# B&R Automation Studio project NAEUL004C00R13L518F00 (part 20)

#### Act_OptP0933PusherConvFB.st
```iecst
ACTION Act_OptP0933PusherConvFB:
//	IF p_bAlarmErr THEN
//		tyP0933PushConv.tyFB.tyBtnStop.bRtCompl := TRUE;
//	END_IF
	//Parameter
	diMnlMtrPshrExtSpd	:= tyP0933PushConv.tyFB.tyNumExtSpd.diValue;
//	diMnlMtrPshrExtTorq	:= tyP0933PushConv.tyFB.tyNumExtTorqPercent.diValue;

	//Pusher Torque & Force Real Time Changing
	//diMnlMtrPshrExtTorq := diConstant1 + (((tyP0933PushConv.tyFB.tyNumExtTorqPercent.diValue -10)/10)*diConstant2/100); //10~30N
//	diMnlMtrPshrExtTorq := p_tyNtParamPPTorqParam.usiStartTorque + (((tyP0933PushConv.tyFB.tyNumExtTorqPercent.diValue -10)/10)*p_tyNtParamPPTorqParam.uiRatio/100); //10~30N
	IF p_tyNtParamCurr.bProjServoPullerPusherPrep THEN
		diMnlMtrPshrExtTorq := p_tyNtParamPPTorqParam.usiStartTorque + (((tyP0933PushConv.tyFB.tyNumExtTorqPercent.diValue -10)/10)*p_tyNtParamPPTorqParam.uiRatio/100); //10~30N
	ELSE
		diMnlMtrPshrExtTorq := tyP0933PushConv.tyFB.tyNumExtTorqPercent.diValue;
	END_IF
	//Conveyor
	IF tyP0933PushConv.tyFB.tyBtnStop.bRtCompl = TRUE THEN
		diMnlPPJogSpd	:= 0;
		ePshrConvAct	:= ConvActPshrRstAll;
//		usiExtRetTest := 0; //Ah Liang

		IF p_ePshrConvStat = ConvActPshrRstAll AND p_ePshrConvStatus = Done THEN
			ePshrConvAct	:= ConvActIdle;

			tyP0933PushConv.tyFB.tyBtnEnt.bRtCompl		:= FALSE;
			tyP0933PushConv.tyFB.tyBtnEnt.bValue		:= FALSE;
			tyP0933PushConv.tyFB.tyBtnEnt.bRtLk			:= FALSE;

			tyP0933PushConv.tyFB.tyBtnExit.bRtCompl		:= FALSE;
			tyP0933PushConv.tyFB.tyBtnExit.bValue		:= FALSE;
			tyP0933PushConv.tyFB.tyBtnExit.bRtLk		:= FALSE;

			tyP0933PushConv.tyFB.tyBtnCylExit.bRtCompl	:= FALSE;
			tyP0933PushConv.tyFB.tyBtnCylExit.bValue	:= FALSE;
			tyP0933PushConv.tyFB.tyBtnCylExit.bRtLk		:= FALSE;

			tyP0933PushConv.tyFB.tyBtnStop.bRtCompl		:= FALSE;
			tyP0933PushConv.tyFB.tyBtnStop.bValue		:= TRUE;
			tyP0933PushConv.tyFB.tyBtnStop.bRtLk		:= TRUE;
		END_IF

	ELSIF tyP0933PushConv.tyFB.tyBtnEnt.bRtCompl = TRUE THEN
		tyP0933PushConv.tyFB.tyBtnEnt.bValue	:= TRUE;
		tyP0933PushConv.tyFB.tyBtnEnt.bRtLk		:= TRUE;

		tyP0933PushConv.tyFB.tyBtnStop.bValue	:= FALSE;
		tyP0933PushConv.tyFB.tyBtnStop.bRtLk	:= FALSE;

		ePshrConvAct	:= ConvActEnt;
		fUIInRtStatOff(ADR(tyP0930MagConv1.tyCom.tyBtnSwitch.uiMaskRtStat));

		IF p_ePshrConvStat = ConvActEnt AND p_ePshrConvStatus = Done THEN
			ePshrConvAct	:= ConvActIdle;

			tyP0933PushConv.tyFB.tyBtnEnt.bRtCompl	:= FALSE;

			tyP0933PushConv.tyFB.tyBtnEnt.bValue	:= FALSE;
			tyP0933PushConv.tyFB.tyBtnEnt.bRtLk		:= FALSE;

			tyP0933PushConv.tyFB.tyBtnStop.bValue	:= TRUE;
			tyP0933PushConv.tyFB.tyBtnStop.bRtLk	:= TRUE;
			fUIInRtStatHide(ADR(tyP0930MagConv1.tyCom.tyBtnSwitch.uiMaskRtStat));
		END_IF

	ELSIF tyP0933PushConv.tyFB.tyBtnExit.bRtCompl = TRUE THEN
		tyP0933PushConv.tyFB.tyBtnExit.bValue	:= TRUE;
		tyP0933PushConv.tyFB.tyBtnExit.bRtLk	:= TRUE;

		tyP0933PushConv.tyFB.tyBtnStop.bValue	:= FALSE;
		tyP0933PushConv.tyFB.tyBtnStop.bRtLk	:= FALSE;

		ePshrConvAct	:= ConvActExit;

		IF p_ePshrConvStat = ConvActExit AND p_ePshrConvStatus = Done THEN
			ePshrConvAct	:= ConvActIdle;

			tyP0933PushConv.tyFB.tyBtnExit.bRtCompl	:= FALSE;

			tyP0933PushConv.tyFB.tyBtnExit.bValue	:= FALSE;
			tyP0933PushConv.tyFB.tyBtnExit.bRtLk	:= FALSE;

			tyP0933PushConv.tyFB.tyBtnStop.bValue	:= TRUE;
			tyP0933PushConv.tyFB.tyBtnStop.bRtLk	:= TRUE;
		END_IF

	ELSIF tyP0933PushConv.tyFB.tyBtnCylExit.bRtCompl = TRUE THEN
		tyP0933PushConv.tyFB.tyBtnCylExit.bValue	:= TRUE;
		tyP0933PushConv.tyFB.tyBtnCylExit.bRtLk		:= TRUE;

		tyP0933PushConv.tyFB.tyBtnStop.bValue		:= FALSE;
		tyP0933PushConv.tyFB.tyBtnStop.bRtLk		:= FALSE;
		diMnlPPJogSpd	:= diMnlMtrPshrExtSpd*diMnlServoMtrMaxPulRatio;
		ePshrConvAct	:= ConvActExitPshr;
		fUIInRtStatOff(ADR(tyP0933PushConv.tyCom.tyBtnSwitch.uiMaskRtStat));

		IF p_ePshrConvStat = ConvActExitPshr AND p_ePshrConvStatus = Done THEN
			ePshrConvAct	:= ConvActIdle;

			tyP0933PushConv.tyFB.tyBtnCylExit.bRtCompl	:= FALSE;

			tyP0933PushConv.tyFB.tyBtnCylExit.bValue	:= FALSE;
			tyP0933PushConv.tyFB.tyBtnCylExit.bRtLk		:= FALSE;

			tyP0933PushConv.tyFB.tyBtnStop.bValue		:= TRUE;
			tyP0933PushConv.tyFB.tyBtnStop.bRtLk		:= TRUE;

		END_IF

	END_IF

	//Pusher
	IF p_tyNtParamCurr.bProjServoPullerPusherPrep = TRUE AND tyP0933PushConv.tyFB.tyBtnStop.bRtCompl = FALSE THEN

		IF tyP0933PushConv.tyCom.tyBtnSwitch.bValue = FALSE THEN
			IF tyP0933PushConv.tyFB.tyBtnRet.bRtCompl = TRUE THEN
				tyP0933PushConv.tyFB.tyBtnRet.bRtCompl	:= FALSE;

				tyP0933PushConv.tyFB.tyBtnRet.bValue	:= TRUE;
				tyP0933PushConv.tyFB.tyBtnExt.bValue	:= FALSE;

			ELSIF tyP0933PushConv.tyFB.tyBtnExt.bRtCompl = TRUE THEN
				tyP0933PushConv.tyFB.tyBtnExt.bRtCompl	:= FALSE;

				tyP0933PushConv.tyFB.tyBtnExt.bValue	:= TRUE;
				tyP0933PushConv.tyFB.tyBtnRet.bValue	:= FALSE;

			END_IF

			IF tyP0933PushConv.tyFB.tyBtnRet.bValue = TRUE THEN
				ePshrConvAct	:= ConvActPshrRet;
				diMnlPPJogSpd	:= diMnlMtrPshrExtSpd*diMnlServoMtrMaxPulRatio;

				tyP0933PushConv.tyFB.tyBtnStop.bValue		:= FALSE;
				tyP0933PushConv.tyFB.tyBtnStop.bRtLk		:= FALSE;

				IF p_ePshrConvStat = ConvActPshrRet AND p_ePshrConvStatus = Done THEN
					ePshrConvAct	:= ConvActIdle;
					diMnlPPJogSpd	:= 0;
					tyP0933PushConv.tyFB.tyBtnRet.bValue	:= FALSE;

				ELSIF p_ePshrConvStatus = Error THEN
					tyP0933PushConv.tyFB.tyBtnRet.bValue	:= FALSE;
					diMnlPPJogSpd	:= 0;
				END_IF

			ELSIF tyP0933PushConv.tyFB.tyBtnExt.bValue = TRUE THEN
				ePshrConvAct	:= ConvActPshrExt;
				diMnlPPJogSpd	:= diMnlMtrPshrExtSpd*diMnlServoMtrMaxPulRatio;
				tyP0933PushConv.tyFB.tyBtnStop.bValue		:= FALSE;
				tyP0933PushConv.tyFB.tyBtnStop.bRtLk		:= FALSE;

				IF p_ePshrConvStat = ConvActPshrExt AND p_ePshrConvStatus = Done THEN
					ePshrConvAct	:= ConvActIdle;
					diMnlPPJogSpd	:= 0;
					tyP0933PushConv.tyFB.tyBtnExt.bValue := FALSE;

				ELSIF p_ePshrConvStatus = Error THEN
					tyP0933PushConv.tyFB.tyBtnExt.bValue := FALSE;
					diMnlPPJogSpd	:= 0;
				END_IF

			END_IF

			//Update Status
			tyP0933PushConv.tyDC.tyBtnRet.bValue	:= NOT p_bPshrConvPshrExtCtrl;
			tyP0933PushConv.tyDC.tyBtnExt.bValue	:= p_bPshrConvPshrExtCtrl;

		END_IF

	ELSIF p_tyNtParamCurr.bProjServoPullerPusherPrep = FALSE AND tyP0933PushConv.tyFB.tyBtnStop.bRtCompl = FALSE
		THEN
//		IF usiExtRetTest = 0 THEN //Ah Liang Start
//			fbPushRetRestTmr(IN:=FALSE);
//			fbPushExtRestTmr(IN:=FALSE);
//		ELSIF usiExtRetTest = 1 THEN
//			fbPushRetRestTmr(IN:=TRUE);
//			fbPushExtRestTmr(IN:=FALSE);
//		ELSIF usiExtRetTest = 2 THEN
//			fbPushExtRestTmr(IN:=TRUE);
//			fbPushRetRestTmr(IN:=FALSE);
//		END_IF
//		IF fbPushRetRestTmr.Q THEN
//			tyP0933PushConv.tyFB.tyBtnExt.bRtCompl := TRUE;
//		ELSIF fbPushExtRestTmr.Q  THEN
//			tyP0933PushConv.tyFB.tyBtnRet.bRtCompl := TRUE;
//		END_IF //Ah Liang End

		IF tyP0933PushConv.tyCom.tyBtnSwitch.bValue = FALSE THEN
			IF tyP0933PushConv.tyFB.tyBtnRet.bRtCompl = TRUE THEN
				tyP0933PushConv.tyFB.tyBtnRet.bRtCompl	:= FALSE;

				tyP0933PushConv.tyFB.tyBtnRet.bValue	:= TRUE;
				tyP0933PushConv.tyFB.tyBtnExt.bValue	:= FALSE;

			ELSIF tyP0933PushConv.tyFB.tyBtnExt.bRtCompl = TRUE THEN
				tyP0933PushConv.tyFB.tyBtnExt.bRtCompl	:= FALSE;

				tyP0933PushConv.tyFB.tyBtnExt.bValue	:= TRUE;
				tyP0933PushConv.tyFB.tyBtnRet.bValue	:= FALSE;

			END_IF

			IF tyP0933PushConv.tyFB.tyBtnRet.bValue = TRUE THEN
				ePshrConvAct	:= ConvActPshrRet;

				tyP0933PushConv.tyFB.tyBtnStop.bValue		:= FALSE;
				tyP0933PushConv.tyFB.tyBtnStop.bRtLk		:= FALSE;

				IF p_ePshrConvStat = ConvActPshrRet AND p_ePshrConvStatus = Done THEN
					ePshrConvAct	:= ConvActIdle;

					tyP0933PushConv.tyFB.tyBtnRet.bValue	:= FALSE;
					//for testing Ah Liang
//					tyP0933PushConv.tyFB.tyBtnExt.bRtCompl := TRUE;
//					usiExtRetTest := 1 ;

				ELSIF p_ePshrConvStatus = Error THEN
					tyP0933PushConv.tyFB.tyBtnRet.bValue	:= FALSE;

				END_IF

			ELSIF tyP0933PushConv.tyFB.tyBtnExt.bValue = TRUE THEN
				ePshrConvAct			:= ConvActPshrExt;

				tyP0933PushConv.tyFB.tyBtnStop.bValue		:= FALSE;
				tyP0933PushConv.tyFB.tyBtnStop.bRtLk		:= FALSE;

				IF p_ePshrConvStat = ConvActPshrExt AND p_ePshrConvStatus = Done THEN
					ePshrConvAct	:= ConvActIdle;

					tyP0933PushConv.tyFB.tyBtnExt.bValue := FALSE;
					//for testing Ah Liang
//					tyP0933PushConv.tyFB.tyBtnRet.bRtCompl := TRUE;
//					usiExtRetTest := 2;
				ELSIF p_ePshrConvStatus = Error THEN
					tyP0933PushConv.tyFB.tyBtnExt.bValue := FALSE;

				END_IF

			END_IF

			//Update Status
			tyP0933PushConv.tyDC.tyBtnRet.bValue	:= NOT p_bPshrConvPshrExtCtrl;
			tyP0933PushConv.tyDC.tyBtnExt.bValue	:= p_bPshrConvPshrExtCtrl;

		END_IF

	ELSE

		tyP0933PushConv.tyFB.tyBtnExt.bRtCompl		:= FALSE;
		tyP0933PushConv.tyFB.tyBtnExt.bValue		:= FALSE;
		tyP0933PushConv.tyFB.tyBtnExt.bRtLk			:= FALSE;

		tyP0933PushConv.tyFB.tyBtnRet.bRtCompl		:= FALSE;
		tyP0933PushConv.tyFB.tyBtnRet.bValue		:= FALSE;
		tyP0933PushConv.tyFB.tyBtnRet.bRtLk			:= FALSE;

	END_IF

	//Pusher
	IF tyP0933PushConv.tyCom.tyBtnSwitch.bValue = FALSE THEN

		IF tyP0933PushConv.tyFB.tyBtnRet.bRtCompl = TRUE THEN
			tyP0933PushConv.tyFB.tyBtnRet.bRtCompl	:= FALSE;

			tyP0933PushConv.tyFB.tyBtnRet.bValue	:= TRUE;
			tyP0933PushConv.tyFB.tyBtnExt.bValue	:= FALSE;

		ELSIF tyP0933PushConv.tyFB.tyBtnExt.bRtCompl = TRUE THEN
			tyP0933PushConv.tyFB.tyBtnExt.bRtCompl	:= FALSE;

			tyP0933PushConv.tyFB.tyBtnExt.bValue	:= TRUE;
			tyP0933PushConv.tyFB.tyBtnRet.bValue	:= FALSE;

		END_IF

		IF tyP0933PushConv.tyFB.tyBtnRet.bValue = TRUE THEN
			ePshrConvAct	:= ConvActPshrRet;

			IF p_ePshrConvStat = ConvActPshrRet AND p_ePshrConvStatus = Done THEN
				ePshrConvAct	:= ConvActIdle;

				tyP0933PushConv.tyFB.tyBtnRet.bValue	:= FALSE;

			ELSIF p_ePshrConvStatus = Error THEN
				tyP0933PushConv.tyFB.tyBtnRet.bValue	:= FALSE;

			END_IF

		ELSIF tyP0933PushConv.tyFB.tyBtnExt.bValue = TRUE THEN
			ePshrConvAct	:= ConvActPshrExt;

			IF p_ePshrConvStat = ConvActPshrExt AND p_ePshrConvStatus = Done THEN
				ePshrConvAct	:= ConvActIdle;

				tyP0933PushConv.tyFB.tyBtnExt.bValue := FALSE;

			ELSIF p_ePshrConvStatus = Error THEN
				tyP0933PushConv.tyFB.tyBtnExt.bValue := FALSE;

			END_IF

		END_IF

		//Update Status
		tyP0933PushConv.tyDC.tyBtnRet.bValue	:= NOT p_bPshrConvPshrExtCtrl;
		tyP0933PushConv.tyDC.tyBtnExt.bValue	:= p_bPshrConvPshrExtCtrl;

	END_IF

	//Mask
	IF p_ePshrConvStatus = Error THEN

		fUIInRtStatOff(ADR(tyP0933PushConv.tyFB.tyBtnEnt.uiMaskRtStat));
		fUIInRtStatOff(ADR(tyP0933PushConv.tyFB.tyBtnExit.uiMaskRtStat));
		fUIInRtStatOff(ADR(tyP0933PushConv.tyFB.tyBtnExt.uiMaskRtStat));
		fUIInRtStatOff(ADR(tyP0933PushConv.tyFB.tyBtnCylExit.uiMaskRtStat));
		fUIInRtStatOff(ADR(tyP0933PushConv.tyFB.tyBtnRet.uiMaskRtStat));
		fUIInRtStatHide(ADR(tyP0933PushConv.tyCom.tyBtnSwitch.uiMaskRtStat));

	ELSIF tyP0933PushConv.tyFB.tyBtnEnt.bRtCompl = TRUE THEN

		fUIInRtStatHide(ADR(tyP0933PushConv.tyFB.tyBtnEnt.uiMaskRtStat));
		fUIInRtStatOff(ADR(tyP0933PushConv.tyFB.tyBtnExit.uiMaskRtStat));
		fUIInRtStatOff(ADR(tyP0933PushConv.tyFB.tyBtnCylExit.uiMaskRtStat));
		fUIInRtStatOff(ADR(tyP0933PushConv.tyFB.tyBtnExt.uiMaskRtStat));
		fUIInRtStatOff(ADR(tyP0933PushConv.tyFB.tyBtnRet.uiMaskRtStat));
		fUIInRtStatOff(ADR(tyP0933PushConv.tyCom.tyBtnSwitch.uiMaskRtStat));

	ELSIF tyP0933PushConv.tyFB.tyBtnExit.bRtCompl = TRUE THEN

		fUIInRtStatOff(ADR(tyP0933PushConv.tyFB.tyBtnEnt.uiMaskRtStat));
		fUIInRtStatHide(ADR(tyP0933PushConv.tyFB.tyBtnExit.uiMaskRtStat));
		fUIInRtStatOff(ADR(tyP0933PushConv.tyFB.tyBtnCylExit.uiMaskRtStat));
		fUIInRtStatOff(ADR(tyP0933PushConv.tyFB.tyBtnExt.uiMaskRtStat));
		fUIInRtStatOff(ADR(tyP0933PushConv.tyFB.tyBtnRet.uiMaskRtStat));
		fUIInRtStatOff(ADR(tyP0933PushConv.tyCom.tyBtnSwitch.uiMaskRtStat));

	ELSIF tyP0933PushConv.tyFB.tyBtnCylExit.bRtCompl = TRUE THEN

		fUIInRtStatOff(ADR(tyP0933PushConv.tyFB.tyBtnEnt.uiMaskRtStat));
		fUIInRtStatOff(ADR(tyP0933PushConv.tyFB.tyBtnExit.uiMaskRtStat));
		fUIInRtStatHide(ADR(tyP0933PushConv.tyFB.tyBtnCylExit.uiMaskRtStat));
		fUIInRtStatOff(ADR(tyP0933PushConv.tyFB.tyBtnExt.uiMaskRtStat));
		fUIInRtStatOff(ADR(tyP0933PushConv.tyFB.tyBtnRet.uiMaskRtStat));
		fUIInRtStatOff(ADR(tyP0933PushConv.tyCom.tyBtnSwitch.uiMaskRtStat));

	ELSIF tyP0933PushConv.tyFB.tyBtnExt.bValue = TRUE OR tyP0933PushConv.tyFB.tyBtnRet.bValue = TRUE THEN

		fUIInRtStatOff(ADR(tyP0933PushConv.tyFB.tyBtnEnt.uiMaskRtStat));
		fUIInRtStatOff(ADR(tyP0933PushConv.tyFB.tyBtnExit.uiMaskRtStat));
		fUIInRtStatHide(ADR(tyP0933PushConv.tyFB.tyBtnExt.uiMaskRtStat));
		fUIInRtStatOff(ADR(tyP0933PushConv.tyFB.tyBtnCylExit.uiMaskRtStat));
		fUIInRtStatHide(ADR(tyP0933PushConv.tyFB.tyBtnRet.uiMaskRtStat));
		fUIInRtStatOff(ADR(tyP0933PushConv.tyCom.tyBtnSwitch.uiMaskRtStat));

	ELSE

		fUIInRtStatHide(ADR(tyP0933PushConv.tyFB.tyBtnEnt.uiMaskRtStat));
		fUIInRtStatHide(ADR(tyP0933PushConv.tyFB.tyBtnExit.uiMaskRtStat));
		fUIInRtStatHide(ADR(tyP0933PushConv.tyFB.tyBtnExt.uiMaskRtStat));
		fUIInRtStatHide(ADR(tyP0933PushConv.tyFB.tyBtnCylExit.uiMaskRtStat));
		fUIInRtStatHide(ADR(tyP0933PushConv.tyFB.tyBtnRet.uiMaskRtStat));
		fUIInRtStatHide(ADR(tyP0933PushConv.tyCom.tyBtnSwitch.uiMaskRtStat));

	END_IF

	IF p_tyNtParamCurr.bProjOutletShutPrep AND NOT(p_tyNtParamCurr.bProjOutletShut2Prep) AND NOT(p_tyNtParamCurr.bProjOutletShut2Prep) THEN//single shutter case
		IF p_bLifterBtmSltAPosDiff OR ((p_bTravDPosDiff AND p_bTravEPosDiff AND p_bTravFPosDiff) OR NOT(p_tyDI.bOutShutterOpenRS) )
			THEN
			fUIInRtStatOff(ADR(tyP0933PushConv.tyFB.tyBtnCylExit.uiMaskRtStat));
			fUIInRtStatOff(ADR(tyP0933PushConv.tyFB.tyBtnExit.uiMaskRtStat));
			fUIInRtStatOff(ADR(tyP0933PushConv.tyFB.tyBtnExt.uiMaskRtStat));
		END_IF
	ELSIF p_tyNtParamCurr.bProjOutletShutPrep AND p_tyNtParamCurr.bProjOutletShut2Prep AND p_tyNtParamCurr.bProjOutletShut2Prep THEN //3 shutter case
		IF p_bLifterBtmSltAPosDiff OR ((p_bTravDPosDiff OR NOT(p_tyDI.bOutShutterOpenRS) ) AND (p_bTravEPosDiff OR NOT(p_tyDI.bOutShutterOpenRS2)) AND (p_bTravFPosDiff OR NOT(p_tyDI.bOutShutterOpenRS3)))
			THEN
			fUIInRtStatOff(ADR(tyP0933PushConv.tyFB.tyBtnCylExit.uiMaskRtStat));
			fUIInRtStatOff(ADR(tyP0933PushConv.tyFB.tyBtnExit.uiMaskRtStat));
			fUIInRtStatOff(ADR(tyP0933PushConv.tyFB.tyBtnExt.uiMaskRtStat));
		END_IF
	END_IF

	//Shutter Control
	IF tyP0933PushConv.tyInOutletShutterFB.tyBtnOpen.bRtCompl = TRUE THEN
		tyP0933PushConv.tyInOutletShutterFB.tyBtnOpen.bRtCompl	:= FALSE;

		tyP0933PushConv.tyInOutletShutterFB.tyBtnOpen.bValue	:= TRUE;
		tyP0933PushConv.tyInOutletShutterFB.tyBtnClose.bValue	:= FALSE;

	ELSIF tyP0933PushConv.tyInOutletShutterFB.tyBtnClose.bRtCompl = TRUE THEN
		tyP0933PushConv.tyInOutletShutterFB.tyBtnClose.bRtCompl	:= FALSE;

		tyP0933PushConv.tyInOutletShutterFB.tyBtnClose.bValue	:= TRUE;
		tyP0933PushConv.tyInOutletShutterFB.tyBtnOpen.bValue	:= FALSE;
	END_IF

	IF tyP0933PushConv.tyInOutletShutterFB.tyBtnOpen.bValue = TRUE THEN
		eInShutterAct	:= PneuActRet;
		eOutShutterAct	:= PneuActRet;

		IF (p_eInShutterStat = PneuActRet AND p_eInShutterStatus = Done)
			AND (p_eOutShutterStat = PneuActRet AND p_eOutShutterStatus = Done)
			THEN
			eInShutterAct	:= PneuActIdle;
			eOutShutterAct	:= PneuActIdle;
			tyP0933PushConv.tyInOutletShutterFB.tyBtnOpen.bValue	:= FALSE;
		ELSIF p_eInShutterStatus = Error OR p_eOutShutterStatus = Error THEN
			tyP0933PushConv.tyInOutletShutterFB.tyBtnOpen.bValue	:= FALSE;
		END_IF

	ELSIF tyP0933PushConv.tyInOutletShutterFB.tyBtnClose.bValue = TRUE THEN
		eInShutterAct	:= PneuActExt;
		eOutShutterAct	:= PneuActExt;
		IF (p_eInShutterStat = PneuActExt AND p_eInShutterStatus = Done)
			AND (p_eOutShutterStat = PneuActExt AND p_eOutShutterStatus = Done)
			THEN
			eInShutterAct	:= PneuActIdle;
			eOutShutterAct	:= PneuActIdle;
			tyP0933PushConv.tyInOutletShutterFB.tyBtnClose.bValue := FALSE;
		ELSIF p_eInShutterStatus = Error OR p_eOutShutterStatus = Error THEN
			tyP0933PushConv.tyInOutletShutterFB.tyBtnClose.bValue := FALSE;
		END_IF
	END_IF

END_ACTION
```

#### Act_OptP0933PusherConvFBStat.st
```iecst
ACTION Act_OptP0933PusherConvFBStat:

	tyP0933PushConv.tyFB.tyStringStat.sValue   := p_sPshrConvStatTxt;

END_ACTION
```

#### Act_OptP0933PusherConvDC.st
```iecst
ACTION Act_OptP0933PusherConvDC:

	//Conveyor
	IF tyP0933PushConv.tyDC.tyBtnStop.bRtCompl = TRUE THEN
		ePshrConvAct	:= ConvActStop;
	//	eMtrPshrAct	:= MtrPshrActStop;

		IF (p_ePshrConvStat = ConvActStop AND p_ePshrConvStatus = Done)
	//		AND	(p_eMtrPshrStat = MtrPshrActStop AND p_eMtrPshrStatus = Done)
			THEN

	//		eMtrPshrAct	:= MtrPshrActIdle;
			ePshrConvAct	:= ConvActIdle;

			tyP0933PushConv.tyDC.tyBtnStop.bRtCompl		:= FALSE;
			tyP0933PushConv.tyDC.tyBtnStop.bValue		:= TRUE;
			tyP0933PushConv.tyDC.tyBtnStop.bRtLk		:= TRUE;

			tyP0933PushConv.tyDC.tyBtnStart.bRtCompl	:= FALSE;
			tyP0933PushConv.tyDC.tyBtnStart.bValue		:= FALSE;
			tyP0933PushConv.tyDC.tyBtnStart.bRtLk		:= FALSE;
		END_IF

	ELSIF tyP0933PushConv.tyDC.tyBtnStart.bRtCompl = TRUE THEN
		tyP0933PushConv.tyDC.tyBtnStart.bValue	:= TRUE;
		tyP0933PushConv.tyDC.tyBtnStart.bRtLk	:= TRUE;

		tyP0933PushConv.tyDC.tyBtnStop.bValue	:= FALSE;
		tyP0933PushConv.tyDC.tyBtnStop.bRtLk	:= FALSE;

		ePshrConvAct	:= ConvActSetMtrSigOnOrLToR;

		IF p_ePshrConvStat = ConvActSetMtrSigOnOrLToR AND p_ePshrConvStatus = Done THEN
			ePshrConvAct	:= ConvActIdle;

			tyP0933PushConv.tyDC.tyBtnStart.bRtCompl	:= FALSE;
		END_IF

	END_IF

	//Pusher
	IF tyP0933PushConv.tyCom.tyBtnSwitch.bValue = TRUE THEN

		IF p_bPshrConvPshrTwoOutputCtrl = FALSE THEN

			IF tyP0933PushConv.tyDC.tyBtnRet.bRtCompl = TRUE THEN
				tyP0933PushConv.tyDC.tyBtnRet.bValue	:= TRUE;
				tyP0933PushConv.tyDC.tyBtnExt.bValue	:= FALSE;

				ePshrConvAct	:= ConvActPshrSetRet;

				IF p_ePshrConvStat = ConvActPshrSetRet AND p_ePshrConvStatus = Done THEN
					ePshrConvAct	:= ConvActIdle;

					tyP0933PushConv.tyDC.tyBtnRet.bRtCompl	:= FALSE;
				END_IF

			ELSIF tyP0933PushConv.tyDC.tyBtnExt.bRtCompl = TRUE THEN
				tyP0933PushConv.tyDC.tyBtnExt.bValue	:= TRUE;
				tyP0933PushConv.tyDC.tyBtnRet.bValue	:= FALSE;

				ePshrConvAct	:= ConvActPshrSetExt;

				IF p_ePshrConvStat = ConvActPshrSetExt AND p_ePshrConvStatus = Done THEN
					ePshrConvAct	:= ConvActIdle;

					tyP0933PushConv.tyDC.tyBtnExt.bRtCompl	:= FALSE;
				END_IF

			END_IF

		ELSE

			IF (tyP0933PushConv.tyDC.tyBtnRet.bRtCompl = TRUE) OR (tyP0933PushConv.tyDC.tyBtnExt.bRtCompl = TRUE) THEN
				IF (tyP0933PushConv.tyDC.tyBtnRet.bValue = TRUE) AND (tyP0933PushConv.tyDC.tyBtnExt.bValue = TRUE) THEN
					ePshrConvAct	:= ConvActPshrSetAll;

					IF p_ePshrConvStat = ConvActPshrSetAll AND p_ePshrConvStatus = Done THEN
						ePshrConvAct	:= ConvActIdle;

						tyP0933PushConv.tyDC.tyBtnRet.bRtCompl	:= FALSE;
						tyP0933PushConv.tyDC.tyBtnExt.bRtCompl	:= FALSE;
					END_IF

				ELSIF (tyP0933PushConv.tyDC.tyBtnRet.bValue = TRUE) AND (tyP0933PushConv.tyDC.tyBtnExt.bValue = FALSE) THEN
					ePshrConvAct	:= ConvActPshrSetRet;

					IF p_ePshrConvStat = ConvActPshrSetRet AND p_ePshrConvStatus = Done THEN
						ePshrConvAct	:= ConvActIdle;

						tyP0933PushConv.tyDC.tyBtnRet.bRtCompl	:= FALSE;
						tyP0933PushConv.tyDC.tyBtnExt.bRtCompl	:= FALSE;
					END_IF

				ELSIF (tyP0933PushConv.tyDC.tyBtnRet.bValue = FALSE) AND (tyP0933PushConv.tyDC.tyBtnExt.bValue = TRUE) THEN
					ePshrConvAct	:= ConvActPshrSetExt;

					IF p_ePshrConvStat = ConvActPshrSetExt AND p_ePshrConvStatus = Done THEN
						ePshrConvAct	:= ConvActIdle;

						tyP0933PushConv.tyDC.tyBtnRet.bRtCompl	:= FALSE;
						tyP0933PushConv.tyDC.tyBtnExt.bRtCompl	:= FALSE;
					END_IF

				ELSE
					ePshrConvAct	:= ConvActPshrRstAll;

					IF p_ePshrConvStat = ConvActPshrRstAll AND p_ePshrConvStatus = Done THEN
						ePshrConvAct	:= ConvActIdle;

						tyP0933PushConv.tyDC.tyBtnRet.bRtCompl	:= FALSE;
						tyP0933PushConv.tyDC.tyBtnExt.bRtCompl	:= FALSE;
					END_IF

				END_IF

			END_IF

		END_IF

		tyP0933PushConv.tyFB.tyBtnExt.bRtCompl	:= FALSE;
		tyP0933PushConv.tyFB.tyBtnExt.bValue	:= FALSE;
		tyP0933PushConv.tyFB.tyBtnRet.bRtCompl	:= FALSE;
		tyP0933PushConv.tyFB.tyBtnRet.bValue	:= FALSE;

	END_IF

	//For Motorized Puller
	IF tyP0933PushConv.tyDC.tyBtnAlarmRst.bRtCompl = TRUE THEN

		IF tyP0933PushConv.tyDC.tyBtnAlarmRst.bValue = TRUE THEN
			eMtrPshrAct	:= MtrPshrActSetAlmRst;

			IF p_eMtrPshrStat = MtrPshrActSetAlmRst AND p_eMtrPshrStatus = Done THEN
				eMtrPshrAct	:= MtrPshrActIdle;

				tyP0933PushConv.tyDC.tyBtnAlarmRst.bRtCompl	:= FALSE;
			END_IF
		ELSE
			eMtrPshrAct	:= MtrPshrActRstAlmRst;

			IF p_eMtrPshrStat = MtrPshrActRstAlmRst AND p_eMtrPshrStatus = Done THEN
				eMtrPshrAct	:= MtrPshrActIdle;

				tyP0933PushConv.tyDC.tyBtnAlarmRst.bRtCompl	:= FALSE;
			END_IF
		END_IF

	ELSIF tyP0933PushConv.tyDC.tyBtnBrake.bRtCompl = TRUE THEN

		IF tyP0933PushConv.tyDC.tyBtnBrake.bValue = TRUE THEN
			eMtrPshrAct	:= MtrPshrActSetBrake;

			IF p_eMtrPshrStat = MtrPshrActSetBrake AND p_eMtrPshrStatus = Done THEN
				eMtrPshrAct	:= MtrPshrActIdle;

				tyP0933PushConv.tyDC.tyBtnBrake.bRtCompl	:= FALSE;
			END_IF
		ELSE
			eMtrPshrAct	:= MtrPshrActRstBrake;

			IF p_eMtrPshrStat = MtrPshrActRstBrake AND p_eMtrPshrStatus = Done THEN
				eMtrPshrAct	:= MtrPshrActIdle;

				tyP0933PushConv.tyDC.tyBtnBrake.bRtCompl	:= FALSE;
			END_IF
		END_IF

	ELSIF tyP0933PushConv.tyDC.tyBtnSigOn.bRtCompl = TRUE THEN

		IF tyP0933PushConv.tyDC.tyBtnSigOn.bValue = TRUE THEN
			eMtrPshrAct	:= MtrPshrActSetSigOn;

			IF p_eMtrPshrStat = MtrPshrActSetSigOn AND p_eMtrPshrStatus = Done THEN
				eMtrPshrAct	:= MtrPshrActIdle;

				tyP0933PushConv.tyDC.tyBtnSigOn.bRtCompl	:= FALSE;
			END_IF
		ELSE
			eMtrPshrAct	:= MtrPshrActRstSigOn;

			IF p_eMtrPshrStat = MtrPshrActRstSigOn AND p_eMtrPshrStatus = Done THEN
				eMtrPshrAct	:= MtrPshrActIdle;

				tyP0933PushConv.tyDC.tyBtnSigOn.bRtCompl	:= FALSE;
			END_IF
		END_IF

	ELSIF tyP0933PushConv.tyDC.tyBtnSpdBinBit0.bRtCompl = TRUE THEN

		IF tyP0933PushConv.tyDC.tyBtnSpdBinBit0.bValue = TRUE THEN
			eMtrPshrAct	:= MtrPshrActSetSpdBit0;

			IF p_eMtrPshrStat = MtrPshrActSetSpdBit0 AND p_eMtrPshrStatus = Done THEN
				eMtrPshrAct	:= MtrPshrActIdle;

				tyP0933PushConv.tyDC.tyBtnSpdBinBit0.bRtCompl	:= FALSE;
			END_IF
		ELSE
			eMtrPshrAct	:= MtrPshrActRstSpdBit0;

			IF p_eMtrPshrStat = MtrPshrActRstSpdBit0 AND p_eMtrPshrStatus = Done THEN
				eMtrPshrAct	:= MtrPshrActIdle;

				tyP0933PushConv.tyDC.tyBtnSpdBinBit0.bRtCompl	:= FALSE;
			END_IF
		END_IF

	ELSIF tyP0933PushConv.tyDC.tyBtnSpdBinBit1.bRtCompl = TRUE THEN

		IF tyP0933PushConv.tyDC.tyBtnSpdBinBit1.bValue = TRUE THEN
			eMtrPshrAct	:= MtrPshrActSetSpdBit1;

			IF p_eMtrPshrStat = MtrPshrActSetSpdBit1 AND p_eMtrPshrStatus = Done THEN
				eMtrPshrAct	:= MtrPshrActIdle;

				tyP0933PushConv.tyDC.tyBtnSpdBinBit1.bRtCompl	:= FALSE;
			END_IF
		ELSE
			eMtrPshrAct	:= MtrPshrActRstSpdBit1;

			IF p_eMtrPshrStat = MtrPshrActRstSpdBit1 AND p_eMtrPshrStatus = Done THEN
				eMtrPshrAct	:= MtrPshrActIdle;

				tyP0933PushConv.tyDC.tyBtnSpdBinBit1.bRtCompl	:= FALSE;
			END_IF
		END_IF

	ELSIF tyP0933PushConv.tyDC.tyBtnSpdBinBit2.bRtCompl = TRUE THEN

		IF tyP0933PushConv.tyDC.tyBtnSpdBinBit2.bValue = TRUE THEN
			eMtrPshrAct	:= MtrPshrActSetSpdBit2;

			IF p_eMtrPshrStat = MtrPshrActSetSpdBit2 AND p_eMtrPshrStatus = Done THEN
				eMtrPshrAct	:= MtrPshrActIdle;

				tyP0933PushConv.tyDC.tyBtnSpdBinBit2.bRtCompl	:= FALSE;
			END_IF
		ELSE
			eMtrPshrAct	:= MtrPshrActRstSpdBit2;

			IF p_eMtrPshrStat = MtrPshrActRstSpdBit2 AND p_eMtrPshrStatus = Done THEN
				eMtrPshrAct	:= MtrPshrActIdle;

				tyP0933PushConv.tyDC.tyBtnSpdBinBit2.bRtCompl	:= FALSE;
			END_IF
		END_IF

	END_IF

	//Mask
	IF p_ePshrConvStatus = Error THEN

		fUIInRtStatOff(ADR(tyP0933PushConv.tyDC.tyBtnStart.uiMaskRtStat));
		fUIInRtStatOff(ADR(tyP0933PushConv.tyDC.tyBtnExt.uiMaskRtStat));
		fUIInRtStatOff(ADR(tyP0933PushConv.tyDC.tyBtnRet.uiMaskRtStat));

	ELSIF tyP0933PushConv.tyDC.tyBtnStart.bValue = TRUE THEN

		fUIInRtStatHide(ADR(tyP0933PushConv.tyDC.tyBtnStart.uiMaskRtStat));
		fUIInRtStatOff(ADR(tyP0933PushConv.tyDC.tyBtnExt.uiMaskRtStat));
		fUIInRtStatOff(ADR(tyP0933PushConv.tyDC.tyBtnRet.uiMaskRtStat));

	ELSE

		fUIInRtStatHide(ADR(tyP0933PushConv.tyDC.tyBtnStart.uiMaskRtStat));
		fUIInRtStatHide(ADR(tyP0933PushConv.tyDC.tyBtnExt.uiMaskRtStat));
		fUIInRtStatHide(ADR(tyP0933PushConv.tyDC.tyBtnRet.uiMaskRtStat));

	END_IF

	//Mask
	//	tyP0933PushConv.tyDC.tyBtnExt.uiMaskRtStat.0		:= NOT(p_eMtrPshrStatus = Error OR tyP0933PushConv.tyDC.tyBtnRet.bValue);
	tyP0933PushConv.tyDC.tyBtnRet.uiMaskRtStat.0		:= NOT(p_eMtrPshrStatus = Error OR tyP0933PushConv.tyDC.tyBtnExt.bValue);
	tyP0933PushConv.tyDC.tyBtnSigOn.uiMaskRtStat.0		:= NOT(p_eMtrPshrStatus = Error);
	tyP0933PushConv.tyDC.tyBtnAlarmRst.uiMaskRtStat.0	:= NOT(p_eMtrPshrStatus = Error);
	tyP0933PushConv.tyDC.tyBtnBrake.uiMaskRtStat.0		:= NOT(p_eMtrPshrStatus = Error);
	tyP0933PushConv.tyDC.tyBtnSpdBinBit0.uiMaskRtStat.0	:= NOT(p_eMtrPshrStatus = Error);
	tyP0933PushConv.tyDC.tyBtnSpdBinBit1.uiMaskRtStat.0	:= NOT(p_eMtrPshrStatus = Error);
	tyP0933PushConv.tyDC.tyBtnSpdBinBit2.uiMaskRtStat.0	:= NOT(p_eMtrPshrStatus = Error);

	IF p_bLifterBtmSltAPosDiff OR (p_bTravDPosDiff AND p_bTravEPosDiff AND p_bTravFPosDiff)
		OR p_eMtrPshrStatus = Error
		THEN
		fUIInRtStatOff(ADR(tyP0933PushConv.tyDC.tyBtnExt.uiMaskRtStat));
	END_IF

END_ACTION
```

#### Act_OptP0933PusherConvRstMnl.st
```iecst
ACTION Act_OptP0933RstMnl:

	IF EDGEPOS((bManualMod = FALSE) OR (p_ePshrConvStatus = Error) OR (p_eMtrPshrStatus = Error))  THEN

		ePshrConvAct	:= ConvActIdle;
		eMtrPshrAct	:= MtrPshrActIdle;

		//FB - Motor
		tyP0933PushConv.tyFB.tyBtnEnt.bRtCompl					:= FALSE;
		tyP0933PushConv.tyFB.tyBtnExit.bRtCompl					:= FALSE;
		tyP0933PushConv.tyFB.tyBtnCylExit.bRtCompl				:= FALSE;
		tyP0933PushConv.tyFB.tyBtnStop.bRtCompl					:= FALSE;

		tyP0933PushConv.tyFB.tyBtnEnt.bValue					:= FALSE;
		tyP0933PushConv.tyFB.tyBtnExit.bValue					:= FALSE;
		tyP0933PushConv.tyFB.tyBtnCylExit.bValue				:= FALSE;
		tyP0933PushConv.tyFB.tyBtnStop.bValue					:= TRUE;

		tyP0933PushConv.tyFB.tyBtnEnt.bRtLk						:= FALSE;
		tyP0933PushConv.tyFB.tyBtnExit.bRtLk					:= FALSE;
		tyP0933PushConv.tyFB.tyBtnCylExit.bRtLk					:= FALSE;
		tyP0933PushConv.tyFB.tyBtnStop.bRtLk					:= TRUE;

		tyP0933PushConv.tyFB.tyBtnEnt.uiMaskRtStat.0			:= TRUE;
		tyP0933PushConv.tyFB.tyBtnExit.uiMaskRtStat.0			:= TRUE;
		tyP0933PushConv.tyFB.tyBtnCylExit.uiMaskRtStat.0		:= TRUE;
		tyP0933PushConv.tyCom.tyBtnSwitch.uiMaskRtStat.0		:= TRUE;

		//FB - Pneu
		tyP0933PushConv.tyFB.tyBtnExt.bRtCompl					:= FALSE;
		tyP0933PushConv.tyFB.tyBtnRet.bRtCompl					:= FALSE;

		tyP0933PushConv.tyFB.tyBtnExt.bValue					:= FALSE;
		tyP0933PushConv.tyFB.tyBtnRet.bValue					:= FALSE;

		tyP0933PushConv.tyFB.tyBtnExt.uiMaskRtStat.0			:= TRUE;
		tyP0933PushConv.tyFB.tyBtnRet.uiMaskRtStat.0			:= TRUE;

		//DC - Motor
		tyP0933PushConv.tyDC.tyBtnStart.bRtCompl				:= FALSE;
		tyP0933PushConv.tyDC.tyBtnStop.bRtCompl					:= FALSE;

		tyP0933PushConv.tyDC.tyBtnStart.bValue					:= FALSE;
		tyP0933PushConv.tyDC.tyBtnStop.bValue					:= TRUE;

		tyP0933PushConv.tyDC.tyBtnStart.bRtLk					:= FALSE;
		tyP0933PushConv.tyDC.tyBtnStop.bRtLk					:= TRUE;

		tyP0933PushConv.tyDC.tyBtnStart.uiMaskRtStat.0			:= TRUE;
		tyP0933PushConv.tyCom.tyBtnSwitch.uiMaskRtStat.0		:= TRUE;

		//DC - Pneu
		tyP0933PushConv.tyDC.tyBtnExt.bRtCompl					:= FALSE;
		tyP0933PushConv.tyDC.tyBtnRet.bRtCompl					:= FALSE;

		tyP0933PushConv.tyDC.tyBtnExt.bValue					:= FALSE;
		tyP0933PushConv.tyDC.tyBtnRet.bValue					:= FALSE;

		tyP0933PushConv.tyDC.tyBtnExt.uiMaskRtStat.0			:= TRUE;
		tyP0933PushConv.tyDC.tyBtnRet.uiMaskRtStat.0			:= TRUE;

		//DC
		tyP0933PushConv.tyDC.tyBtnExt.bRtCompl			:= FALSE;
		tyP0933PushConv.tyDC.tyBtnRet.bRtCompl			:= FALSE;
		tyP0933PushConv.tyDC.tyBtnSpdBinBit0.bRtCompl	:= FALSE;
		tyP0933PushConv.tyDC.tyBtnSpdBinBit1.bRtCompl	:= FALSE;
		tyP0933PushConv.tyDC.tyBtnSpdBinBit2.bRtCompl	:= FALSE;
		tyP0933PushConv.tyDC.tyBtnSigOn.bRtCompl		:= FALSE;
		tyP0933PushConv.tyDC.tyBtnBrake.bRtCompl		:= FALSE;
		tyP0933PushConv.tyDC.tyBtnAlarmRst.bRtCompl		:= FALSE;

		tyP0933PushConv.tyDC.tyBtnExt.bValue			:= FALSE;
		tyP0933PushConv.tyDC.tyBtnRet.bValue			:= FALSE;
		tyP0933PushConv.tyDC.tyBtnSpdBinBit0.bValue		:= FALSE;
		tyP0933PushConv.tyDC.tyBtnSpdBinBit1.bValue		:= FALSE;
		tyP0933PushConv.tyDC.tyBtnSpdBinBit2.bValue		:= FALSE;
		tyP0933PushConv.tyDC.tyBtnSigOn.bValue			:= FALSE;
		tyP0933PushConv.tyDC.tyBtnBrake.bValue			:= FALSE;
		tyP0933PushConv.tyDC.tyBtnAlarmRst.bValue		:= FALSE;

	END_IF

	IF EDGEPOS(bManualMod = FALSE) THEN
		tyP0933PushConv.tyCom.tyBtnSwitch.bValue := FALSE;

		fUIInRtStatHide(ADR(tyP0933PushConv.tyDC.tyLyr.uiRtStat));
		fUIInRtStatOff(ADR(tyP0933PushConv.tyFB.tyLyr.uiRtStat));

	END_IF

	eInShutterAct	:= PneuActIdle;
	eOutShutterAct	:= PneuActIdle;

	tyP0933PushConv.tyInOutletShutterFB.tyBtnClose.bRtCompl	:= FALSE;
	tyP0933PushConv.tyInOutletShutterFB.tyBtnClose.bValue	:= FALSE;
	tyP0933PushConv.tyInOutletShutterFB.tyBtnOpen.bRtCompl	:= FALSE;
	tyP0933PushConv.tyInOutletShutterFB.tyBtnOpen.bValue	:= FALSE;

END_ACTION
```

#### Act_EntP0934Disp.st
```iecst
ACTION Act_EntP0934Disp:

	//Access Address
	p_tyC0001MotionStd ACCESS ADR(tyP0934AW.tyMotionStd);

	p_tyC0002FullMask ACCESS ADR(tyP0934AW.tyFullMaskHide);

	p_tyC0004Navi ACCESS ADR(tyP0934AW.tyNaviBack);

	p_tyC0005Main ACCESS ADR(tyCommon.tyMain);

	p_tyC0007Notif ACCESS ADR(tyCommon.tyNotif);

	p_tyC0008MsgBox ACCESS ADR(tyP0934AW.tyMsgBoxHide);

	p_tyC0009Info ACCESS ADR(tyCommon.tyInfo);

	p_tyP0934AW ACCESS ADR(tyP0934AW.tyAW);

	p_tyP0934InOutletShutterFB ACCESS ADR(tyP0934AW.tyInOutletShutterFB);

	//Display
	tyP0934AW.tyAW.tyNumNewWidth.diValue	:= p_tyProdRcpCurrRcp0.diWidthInUM;

	tyP0934AW.tyMotionStd.tyBtnPwr.bValue	:= p_bAWOpenPwrOn;

END_ACTION
```

#### Act_OptP0934Navi.st
```iecst
ACTION Act_OptP0934Navi:

	IF tyP0934AW.tyNaviBack.tyBtnBack.bRtCompl = TRUE THEN
		tyP0934AW.tyNaviBack.tyBtnBack.bRtCompl	:= FALSE;
		tyP0934AW.tyNaviBack.tyBtnBack.bValue	:= FALSE;

		eChgPage	:= UIP0920MtrNPneuCtrl;
	END_IF

END_ACTION
```

#### Act_OptP0934FullMask.st
```iecst
ACTION Act_OptP0934FullMask:

	IF eCurrPage = UIP0934AW THEN

		IF p_tyDI.bEStopSig = FALSE THEN
			p_tyC0002FullMask ACCESS ADR(tyP0934AW.tyFullMaskEStop);

		ELSIF p_tyDI.bCoverSWSig = FALSE THEN
			p_tyC0002FullMask ACCESS ADR(tyP0934AW.tyFullMaskCWSig);

		ELSIF p_tyDI.bSafetyRlySig = FALSE THEN
			p_tyC0002FullMask ACCESS ADR(tyP0934AW.tyFullMaskSafetyRly);

		ELSIF p_tyDI.bConvLftSen THEN
			p_tyC0002FullMask ACCESS ADR(tyP0934AW.tyFullMaskLftSenInterrupt);

		ELSIF p_tyDI.bConvMidSen THEN
			p_tyC0002FullMask ACCESS ADR(tyP0934AW.tyFullMaskMidSenInterrupt);

		ELSIF p_tyDI.bConvRgtSen THEN
			p_tyC0002FullMask ACCESS ADR(tyP0934AW.tyFullMaskRgtSenInterrupt);

		ELSIF p_tyDI.bConvClrSen THEN
			p_tyC0002FullMask ACCESS ADR(tyP0934AW.tyFullMaskClrSenInterrupt);

		ELSIF (p_tyNtParamCurr.bProjInletShutPrep AND p_tyDI.bInShutterCloseRS = FALSE) AND NOT(bBypassShutForCalib) THEN
			p_tyC0002FullMask ACCESS ADR(tyP0934AW.tyFullMaskInShutOpnInterrupt);

		ELSIF ((p_tyDI.bOutShutterCloseRS = FALSE AND p_tyNtParamCurr.bProjOutletShutPrep) OR (p_tyDI.bOutShutterCloseRS2 = FALSE AND p_tyNtParamCurr.bProjOutletShut2Prep )OR (p_tyDI.bOutShutterCloseRS3 = FALSE AND p_tyNtParamCurr.bProjOutletShut3Prep)) AND NOT(bBypassShutForCalib) THEN
//			IF p_tyNtParamCurr.bCurtainSenPrep THEN
//				IF (p_tyDI.bOutShutterCloseRS = FALSE AND p_tyNtParamCurr.bProjOutletShutPrep ) OR (p_tyDI.bOutShutterCloseRS2 = FALSE AND p_tyNtParamCurr.bProjOutletShut2Prep)OR (p_tyDI.bOutShutterCloseRS3 = FALSE AND p_tyNtParamCurr.bProjOutletShut3Prep )THEN
//					p_tyC0002FullMask ACCESS ADR(tyP0934AW.tyFullMaskOutShutOpnInterrupt);
//				END_IF
//			ELSE
//				IF p_tyDI.bOutShutterCloseRS = FALSE THEN
					p_tyC0002FullMask ACCESS ADR(tyP0934AW.tyFullMaskOutShutOpnInterrupt);
//				END_IF
//			END_IF
		ELSE
			p_tyC0002FullMask ACCESS ADR(tyP0934AW.tyFullMaskHide);

		END_IF

	END_IF

END_ACTION
```

#### Act_OptP0934FBCtrl.st
```iecst
ACTION Act_OptP0934FBCtrl:

	fbJogSlowToFastDlyTm.PT	:= T#2s;
	fbJogSlowToFastDlyTm;
	fbLmtRstTm;

	//Conveyor Sensor Interruption
	IF (p_tyDI.bConvLftSen OR p_tyDI.bConvMidSen OR p_tyDI.bConvRgtSen OR p_tyDI.bConvClrSen OR p_tyDI.bPusherRetRS = FALSE)
		AND eCurrPage = UIP0934AW
		THEN
		tyP0934AW.tyMotionStd.tyBtnStop.bRtCompl	:= TRUE;
	END_IF

//	IF EDGEPOS((p_udiAWOpenAxisErrID = 21570 OR p_udiAWOpenAxisErrID = 21571)
	IF EDGEPOS((p_bAWOpenFwdLmtSen OR p_bAWOpenRevLmtSen OR p_udiAWOpenAxisErrID = 21570 OR p_udiAWOpenAxisErrID = 21571)
		AND tyP0934AW.tyMotionStd.tyBtnJogOpen.bValue = FALSE
		AND tyP0934AW.tyMotionStd.tyBtnJogClose.bValue = FALSE)
	THEN
		fbLmtRstTm.IN	:= TRUE;
	END_IF

	IF fbLmtRstTm.Q = TRUE THEN
		tyP0934AW.tyMotionStd.tyBtnRst.bRtCompl		:= TRUE;
	END_IF

	IF (tyP0934AW.tyMotionStd.tyBtnJogOpen.bValue = FALSE AND tyP0934AW.tyMotionStd.tyBtnJogClose.bValue = FALSE) AND (p_bAWOpenJogging = TRUE) THEN
		bJogStopAW	:= TRUE;
	END_IF

	IF tyP0934AW.tyMotionStd.tyBtnStop.bRtCompl = TRUE THEN
		eAWOpenAct		:= AWActStop;

		IF p_eAWOpenStat = AWActStop AND p_eAWOpenStatus = Done THEN
			eAWOpenAct	:= AWActIdle;

			tyP0934AW.tyMotionStd.tyBtnStop.bRtCompl			:= FALSE;
			tyP0934AW.tyMotionStd.tyBtnJogOpen.bRtCompl			:= FALSE;
			tyP0934AW.tyMotionStd.tyBtnJogClose.bRtCompl		:= FALSE;
			tyP0934AW.tyMotionStd.tyBtnOrigin.bRtCompl			:= FALSE;
			tyP0934AW.tyMotionStd.tyBtnMovAbs.bRtCompl			:= FALSE;
			tyP0934AW.tyMotionStd.tyBtnMovRel.bRtCompl			:= FALSE;
			tyP0934AW.tyAW.tyBtnGo.bRtCompl						:= FALSE;

			tyP0934AW.tyMotionStd.tyBtnStop.bValue				:= TRUE;
			tyP0934AW.tyMotionStd.tyBtnJogOpen.bValue			:= FALSE;
			tyP0934AW.tyMotionStd.tyBtnJogClose.bValue			:= FALSE;
			tyP0934AW.tyMotionStd.tyBtnOrigin.bValue			:= FALSE;
			tyP0934AW.tyMotionStd.tyBtnMovAbs.bValue			:= FALSE;
			tyP0934AW.tyMotionStd.tyBtnMovRel.bValue			:= FALSE;
			tyP0934AW.tyAW.tyBtnGo.bValue						:= FALSE;

			tyP0934AW.tyMotionStd.tyBtnStop.bRtLk				:= TRUE;
			tyP0934AW.tyMotionStd.tyBtnJogOpen.bRtLk			:= FALSE;
			tyP0934AW.tyMotionStd.tyBtnJogClose.bRtLk			:= FALSE;
			tyP0934AW.tyMotionStd.tyBtnOrigin.bRtLk				:= FALSE;
			tyP0934AW.tyMotionStd.tyBtnMovAbs.bRtLk				:= FALSE;
			tyP0934AW.tyMotionStd.tyBtnMovRel.bRtLk				:= FALSE;
			tyP0934AW.tyAW.tyBtnGo.bRtLk						:= FALSE;
		END_IF

	ELSIF (tyP0934AW.tyMotionStd.tyBtnJogOpen.bRtCompl = TRUE) OR (tyP0934AW.tyMotionStd.tyBtnJogClose.bRtCompl = TRUE) OR (bJogStopAW = TRUE) THEN
		bJogSlow					:= FALSE;
		bJogFast					:= FALSE;
		fbJogSlowToFastDlyTm.IN		:= FALSE;

		eAWOpenAct		:= AWActJogStop;

		IF p_eAWOpenStat = AWActJogStop AND p_eAWOpenStatus = Done THEN
			eAWOpenAct	:= AWActIdle;

			bJogStopAW	:= FALSE;

			tyP0934AW.tyMotionStd.tyBtnStop.bRtCompl		:= FALSE;
			tyP0934AW.tyMotionStd.tyBtnJogOpen.bRtCompl		:= FALSE;
			tyP0934AW.tyMotionStd.tyBtnJogClose.bRtCompl	:= FALSE;
			tyP0934AW.tyMotionStd.tyBtnOrigin.bRtCompl		:= FALSE;
			tyP0934AW.tyMotionStd.tyBtnMovAbs.bRtCompl		:= FALSE;
			tyP0934AW.tyMotionStd.tyBtnMovRel.bRtCompl		:= FALSE;
			tyP0934AW.tyAW.tyBtnGo.bRtCompl					:= FALSE;

			tyP0934AW.tyMotionStd.tyBtnStop.bValue			:= TRUE;
			tyP0934AW.tyMotionStd.tyBtnJogOpen.bValue		:= FALSE;
			tyP0934AW.tyMotionStd.tyBtnJogClose.bValue		:= FALSE;
			tyP0934AW.tyMotionStd.tyBtnOrigin.bValue		:= FALSE;
			tyP0934AW.tyMotionStd.tyBtnMovAbs.bValue		:= FALSE;
			tyP0934AW.tyMotionStd.tyBtnMovRel.bValue		:= FALSE;
			tyP0934AW.tyAW.tyBtnGo.bValue					:= FALSE;

			tyP0934AW.tyMotionStd.tyBtnStop.bRtLk			:= TRUE;
			tyP0934AW.tyMotionStd.tyBtnJogOpen.bRtLk		:= FALSE;
			tyP0934AW.tyMotionStd.tyBtnJogClose.bRtLk		:= FALSE;
			tyP0934AW.tyMotionStd.tyBtnOrigin.bRtLk			:= FALSE;
			tyP0934AW.tyMotionStd.tyBtnMovAbs.bRtLk			:= FALSE;
			tyP0934AW.tyMotionStd.tyBtnMovRel.bRtLk			:= FALSE;
			tyP0934AW.tyAW.tyBtnGo.bRtLk					:= FALSE;
		END_IF

	ELSIF tyP0934AW.tyMotionStd.tyBtnPwr.bRtCompl = TRUE THEN
		tyP0934AW.tyMotionStd.tyBtnPwr.bRtLk					:= TRUE;

		IF tyP0934AW.tyMotionStd.tyBtnPwr.bValue = TRUE THEN
			eAWOpenAct		:= AWActPwrOn;

			IF p_eAWOpenStat = AWActPwrOn AND p_eAWOpenStatus = Done THEN
				eAWOpenAct	:= AWActIdle;

				tyP0934AW.tyMotionStd.tyBtnPwr.bRtCompl			:= FALSE;
				tyP0934AW.tyMotionStd.tyBtnPwr.bRtLk			:= FALSE;
			END_IF
		ELSE
			eAWOpenAct		:= AWActPwrOff;

			IF p_eAWOpenStat = AWActPwrOff AND p_eAWOpenStatus = Done THEN
				eAWOpenAct	:= AWActIdle;

				tyP0934AW.tyMotionStd.tyBtnPwr.bRtCompl			:= FALSE;
				tyP0934AW.tyMotionStd.tyBtnPwr.bRtLk			:= FALSE;
			END_IF
		END_IF

	ELSIF tyP0934AW.tyMotionStd.tyBtnOrigin.bRtCompl = TRUE THEN
		tyP0934AW.tyMotionStd.tyBtnOrigin.bValue				:= TRUE;
		tyP0934AW.tyMotionStd.tyBtnStop.bValue					:= FALSE;

		tyP0934AW.tyMotionStd.tyBtnOrigin.bRtLk					:= TRUE;
		tyP0934AW.tyMotionStd.tyBtnStop.bRtLk					:= FALSE;

		eAWOpenAct		:= AWActHoming;

		IF p_eAWOpenStat = AWActHoming AND p_eAWOpenStatus = Done THEN
			eAWOpenAct	:= AWActIdle;

			tyP0934AW.tyMotionStd.tyBtnOrigin.bRtCompl			:= FALSE;
			tyP0934AW.tyMotionStd.tyBtnOrigin.bValue			:= FALSE;
			tyP0934AW.tyMotionStd.tyBtnStop.bValue				:= TRUE;

			tyP0934AW.tyMotionStd.tyBtnOrigin.bRtLk				:= FALSE;
			tyP0934AW.tyMotionStd.tyBtnStop.bRtLk				:= TRUE;
		END_IF

	ELSIF tyP0934AW.tyMotionStd.tyBtnRst.bRtCompl = TRUE THEN
		tyP0934AW.tyMotionStd.tyBtnRst.bValue					:= TRUE;
		tyP0934AW.tyMotionStd.tyBtnRst.bRtLk					:= TRUE;

		eAWOpenAct		:= AWActRstAxisErr;

		IF p_eAWOpenStat = AWActRstAxisErr AND p_eAWOpenStatus = Done THEN
			eAWOpenAct	:= AWActIdle;

			tyP0934AW.tyMotionStd.tyBtnRst.bRtCompl				:= FALSE;
			tyP0934AW.tyMotionStd.tyBtnRst.bValue				:= FALSE;
			tyP0934AW.tyMotionStd.tyBtnRst.bRtLk				:= FALSE;

			fbLmtRstTm.IN			:= FALSE;
		END_IF

	ELSIF tyP0934AW.tyAW.tyBtnGo.bRtCompl = TRUE THEN
		tyP0934AW.tyAW.tyBtnGo.bValue							:= TRUE;
		tyP0934AW.tyMotionStd.tyBtnStop.bValue					:= FALSE;

		tyP0934AW.tyAW.tyBtnGo.bRtLk							:= TRUE;
		tyP0934AW.tyMotionStd.tyBtnStop.bRtLk					:= FALSE;

		diMnlAWGoWidth		:= tyP0934AW.tyAW.tyNumNewWidth.diValue;
		diMnlAWNomSpd		:= tyP0934AW.tyMotionStd.tyNumNomSpd.diValue;

		eAWOpenAct		:= AWActGoWidth;

		IF p_eAWOpenStat = AWActGoWidth AND p_eAWOpenStatus = Done THEN
			eAWOpenAct	:= AWActIdle;

			tyP0934AW.tyAW.tyBtnGo.bRtCompl						:= FALSE;
			tyP0934AW.tyAW.tyBtnGo.bValue						:= FALSE;
			tyP0934AW.tyMotionStd.tyBtnStop.bValue				:= TRUE;

			tyP0934AW.tyAW.tyBtnGo.bRtLk						:= FALSE;
			tyP0934AW.tyMotionStd.tyBtnStop.bRtLk				:= TRUE;
		END_IF

	ELSIF tyP0934AW.tyMotionStd.tyBtnMovAbs.bRtCompl = TRUE THEN
		tyP0934AW.tyMotionStd.tyBtnMovAbs.bValue				:= TRUE;
		tyP0934AW.tyMotionStd.tyBtnStop.bValue					:= FALSE;

		tyP0934AW.tyMotionStd.tyBtnMovAbs.bRtLk					:= TRUE;
		tyP0934AW.tyMotionStd.tyBtnStop.bRtLk					:= FALSE;

		diMnlAWTargetPos	:= tyP0934AW.tyMotionStd.tyNumTargetPos.diValue;
		diMnlAWNomSpd		:= tyP0934AW.tyMotionStd.tyNumNomSpd.diValue;

		eAWOpenAct		:= AWActMovAbs;

		IF p_eAWOpenStat = AWActMovAbs AND p_eAWOpenStatus = Done THEN
			eAWOpenAct	:= AWActIdle;

			tyP0934AW.tyMotionStd.tyBtnMovAbs.bRtCompl			:= FALSE;
			tyP0934AW.tyMotionStd.tyBtnMovAbs.bValue			:= FALSE;
			tyP0934AW.tyMotionStd.tyBtnStop.bValue				:= TRUE;

			tyP0934AW.tyMotionStd.tyBtnMovAbs.bRtLk				:= FALSE;
			tyP0934AW.tyMotionStd.tyBtnStop.bRtLk				:= TRUE;
		END_IF

	ELSIF tyP0934AW.tyMotionStd.tyBtnMovRel.bRtCompl = TRUE THEN
		tyP0934AW.tyMotionStd.tyBtnMovRel.bValue				:= TRUE;
		tyP0934AW.tyMotionStd.tyBtnStop.bValue					:= FALSE;

		tyP0934AW.tyMotionStd.tyBtnMovRel.bRtLk					:= TRUE;
		tyP0934AW.tyMotionStd.tyBtnStop.bRtLk					:= FALSE;

		diMnlAWStepSize		:= tyP0934AW.tyMotionStd.tyNumStepSize.diValue;
		diMnlAWNomSpd		:= tyP0934AW.tyMotionStd.tyNumNomSpd.diValue;

		eAWOpenAct		:= AWActMovRel;

		IF p_eAWOpenStat = AWActMovRel AND p_eAWOpenStatus = Done THEN
			eAWOpenAct	:= AWActIdle;

			tyP0934AW.tyMotionStd.tyBtnMovRel.bRtCompl			:= FALSE;
			tyP0934AW.tyMotionStd.tyBtnMovRel.bValue			:= FALSE;
			tyP0934AW.tyMotionStd.tyBtnStop.bValue				:= TRUE;

			tyP0934AW.tyMotionStd.tyBtnMovRel.bRtLk				:= FALSE;
			tyP0934AW.tyMotionStd.tyBtnStop.bRtLk				:= TRUE;
		END_IF

	ELSIF (tyP0934AW.tyMotionStd.tyBtnJogOpen.bValue = TRUE) AND (fbJogSlowToFastDlyTm.Q = FALSE) AND (bJogSlow = FALSE) THEN
		tyP0934AW.tyMotionStd.tyBtnStop.bValue					:= FALSE;
		tyP0934AW.tyMotionStd.tyBtnStop.bRtLk					:= FALSE;

		fbJogSlowToFastDlyTm.IN		:= TRUE;

		diMnlAWJogSpd		:= tyP0934AW.tyMotionStd.tyNumSlwSpd.diValue;

		eAWOpenAct		:= AWActJogOpen;

		IF p_eAWOpenStat = AWActJogOpen AND p_eAWOpenStatus = Done THEN
			eAWOpenAct	:= AWActIdle;
			bJogSlow				:= TRUE;
		ELSIF p_eAWOpenStatus = Error THEN
			fbJogSlowToFastDlyTm.IN	:= FALSE;
			bJogSlow				:= TRUE;
		END_IF

	ELSIF (tyP0934AW.tyMotionStd.tyBtnJogOpen.bValue = TRUE) AND (fbJogSlowToFastDlyTm.Q = TRUE) AND (bJogFast = FALSE) THEN
		tyP0934AW.tyMotionStd.tyBtnStop.bValue					:= FALSE;
		tyP0934AW.tyMotionStd.tyBtnStop.bRtLk					:= FALSE;

		fbJogSlowToFastDlyTm.IN		:= TRUE;

		diMnlAWJogSpd		:= tyP0934AW.tyMotionStd.tyNumNomSpd.diValue;

		eAWOpenAct		:= AWActJogOpen;

		IF p_eAWOpenStat = AWActJogOpen AND p_eAWOpenStatus = Done THEN
			eAWOpenAct	:= AWActIdle;
			bJogFast				:= TRUE;
		ELSIF p_eAWOpenStatus = Error THEN
			fbJogSlowToFastDlyTm.IN	:= FALSE;
			bJogFast				:= TRUE;
		END_IF

	ELSIF (tyP0934AW.tyMotionStd.tyBtnJogClose.bValue = TRUE) AND (fbJogSlowToFastDlyTm.Q = FALSE) AND (bJogSlow = FALSE) THEN
		tyP0934AW.tyMotionStd.tyBtnStop.bValue					:= FALSE;
		tyP0934AW.tyMotionStd.tyBtnStop.bRtLk					:= FALSE;

		fbJogSlowToFastDlyTm.IN		:= TRUE;

		diMnlAWJogSpd		:= tyP0934AW.tyMotionStd.tyNumSlwSpd.diValue;

		eAWOpenAct		:= AWActJogClose;

		IF p_eAWOpenStat = AWActJogClose AND p_eAWOpenStatus = Done THEN
			eAWOpenAct	:= AWActIdle;
			bJogSlow				:= TRUE;
		ELSIF p_eAWOpenStatus = Error THEN
			fbJogSlowToFastDlyTm.IN	:= FALSE;
			bJogSlow				:= TRUE;
		END_IF

	ELSIF (tyP0934AW.tyMotionStd.tyBtnJogClose.bValue = TRUE) AND (fbJogSlowToFastDlyTm.Q = TRUE) AND (bJogFast = FALSE) THEN
		tyP0934AW.tyMotionStd.tyBtnStop.bValue					:= FALSE;
		tyP0934AW.tyMotionStd.tyBtnStop.bRtLk					:= FALSE;

		fbJogSlowToFastDlyTm.IN		:= TRUE;

		diMnlAWJogSpd		:= tyP0934AW.tyMotionStd.tyNumNomSpd.diValue;

		eAWOpenAct		:= AWActJogClose;

		IF p_eAWOpenStat = AWActJogClose AND p_eAWOpenStatus = Done THEN
			eAWOpenAct	:= AWActIdle;
			bJogFast				:= TRUE;
		ELSIF p_eAWOpenStatus = Error THEN
			fbJogSlowToFastDlyTm.IN	:= FALSE;
			bJogFast				:= TRUE;
		END_IF
	END_IF

	//Shutter Control
	IF tyP0934AW.tyInOutletShutterFB.tyBtnOpen.bRtCompl = TRUE THEN
		tyP0934AW.tyInOutletShutterFB.tyBtnOpen.bRtCompl	:= FALSE;

		tyP0934AW.tyInOutletShutterFB.tyBtnOpen.bValue	:= TRUE;
		tyP0934AW.tyInOutletShutterFB.tyBtnClose.bValue	:= FALSE;

	ELSIF tyP0934AW.tyInOutletShutterFB.tyBtnClose.bRtCompl = TRUE THEN
		tyP0934AW.tyInOutletShutterFB.tyBtnClose.bRtCompl	:= FALSE;

		tyP0934AW.tyInOutletShutterFB.tyBtnClose.bValue	:= TRUE;
		tyP0934AW.tyInOutletShutterFB.tyBtnOpen.bValue	:= FALSE;
	END_IF

	IF tyP0934AW.tyInOutletShutterFB.tyBtnOpen.bValue = TRUE THEN
		eInShutterAct	:= PneuActRet;
		eOutShutterAct	:= PneuActRet;

		IF (p_eInShutterStat = PneuActRet AND p_eInShutterStatus = Done)
			AND (p_eOutShutterStat = PneuActRet AND p_eOutShutterStatus = Done)
			THEN
			eInShutterAct	:= PneuActIdle;
			eOutShutterAct	:= PneuActIdle;
			tyP0934AW.tyInOutletShutterFB.tyBtnOpen.bValue	:= FALSE;
		ELSIF p_eInShutterStatus = Error OR p_eOutShutterStatus = Error THEN
			tyP0934AW.tyInOutletShutterFB.tyBtnOpen.bValue	:= FALSE;
		END_IF

	ELSIF tyP0934AW.tyInOutletShutterFB.tyBtnClose.bValue = TRUE THEN
		eInShutterAct	:= PneuActExt;
		eOutShutterAct	:= PneuActExt;
		IF (p_eInShutterStat = PneuActExt AND p_eInShutterStatus = Done)
			AND (p_eOutShutterStat = PneuActExt AND p_eOutShutterStatus = Done)
			THEN
			eInShutterAct	:= PneuActIdle;
			eOutShutterAct	:= PneuActIdle;
			tyP0934AW.tyInOutletShutterFB.tyBtnClose.bValue := FALSE;
		ELSIF p_eInShutterStatus = Error OR p_eOutShutterStatus = Error THEN
			tyP0934AW.tyInOutletShutterFB.tyBtnClose.bValue := FALSE;
		END_IF
	END_IF

END_ACTION
```

#### Act_OptP0934FBStat.st
```iecst
ACTION Act_OptP0934FBStat:

	IF p_bAWOpenAxisErr = TRUE THEN
		tyP0934AW.tyMotionStd.tyStringStat.sValue	:= p_sAWOpenAxisErrTxt;
	ELSE
		IF NOT(p_bAWOpenJogging AND p_eAWOpenStat = AWActIdle) THEN
			tyP0934AW.tyMotionStd.tyStringStat.sValue	:= p_sAWOpenStatTxt;
		END_IF
	END_IF

END_ACTION
```

#### Act_OptP0934Mask.st
```iecst
ACTION Act_OptP0934Mask:

	// Interlock Power
	IF p_bAWOpenAxisErr = TRUE AND p_bAWOpenPwrOn = FALSE THEN
		fUIInRtStatOff(ADR(tyP0934AW.tyMotionStd.tyBtnPwr.uiMaskRtStat));
		tyP0934AW.tyMotionStd.tyBtnPwr.bValue		:= FALSE;
	ELSE
		fUIInRtStatHide(ADR(tyP0934AW.tyMotionStd.tyBtnPwr.uiMaskRtStat));
	END_IF

	// Interlock Others Move
	IF p_bAWOpenAxisErr = TRUE OR p_bAWOpenPwrOn = FALSE THEN
		fUIInRtStatOff(ADR(tyP0934AW.tyMotionStd.tyBtnOrigin.uiMaskRtStat));
		fUIInRtStatOff(ADR(tyP0934AW.tyMotionStd.tyBtnMovRel.uiMaskRtStat));
		fUIInRtStatOff(ADR(tyP0934AW.tyMotionStd.tyBtnJogOpen.uiMaskRtStat));
		fUIInRtStatOff(ADR(tyP0934AW.tyMotionStd.tyBtnJogClose.uiMaskRtStat));
	ELSE
		fUIInRtStatHide(ADR(tyP0934AW.tyMotionStd.tyBtnOrigin.uiMaskRtStat));
		fUIInRtStatHide(ADR(tyP0934AW.tyMotionStd.tyBtnMovRel.uiMaskRtStat));
		fUIInRtStatHide(ADR(tyP0934AW.tyMotionStd.tyBtnJogOpen.uiMaskRtStat));
		fUIInRtStatHide(ADR(tyP0934AW.tyMotionStd.tyBtnJogClose.uiMaskRtStat));
	END_IF

	// Interlock Move Absolute
	IF p_bAWOpenAxisErr = TRUE OR p_bAWOpenPwrOn = FALSE OR p_bAWOpenIsHomed = FALSE THEN
		fUIInRtStatOff(ADR(tyP0934AW.tyAW.tyBtnGo.uiMaskRtStat));
		fUIInRtStatOff(ADR(tyP0934AW.tyMotionStd.tyBtnMovAbs.uiMaskRtStat));
	ELSE
		fUIInRtStatHide(ADR(tyP0934AW.tyAW.tyBtnGo.uiMaskRtStat));
		fUIInRtStatHide(ADR(tyP0934AW.tyMotionStd.tyBtnMovAbs.uiMaskRtStat));
	END_IF

	//Interlock Limit Sensor
	IF tyP0934AW.tyMotionStd.tyBtnOpenLmtSen.bValue = TRUE THEN
		fUIInRtStatOff(ADR(tyP0934AW.tyMotionStd.tyBtnJogOpen.uiMaskRtStat));
	END_IF

	IF tyP0934AW.tyMotionStd.tyBtnCloseLmtSen.bValue = TRUE THEN
		fUIInRtStatOff(ADR(tyP0934AW.tyMotionStd.tyBtnJogClose.uiMaskRtStat));
	END_IF

	// Interlock When Moving
	IF tyP0934AW.tyMotionStd.tyBtnOrigin.bRtCompl = TRUE THEN
		fUIInRtStatOff(ADR(tyP0934AW.tyMotionStd.tyBtnMovAbs.uiMaskRtStat));
		fUIInRtStatOff(ADR(tyP0934AW.tyMotionStd.tyBtnMovRel.uiMaskRtStat));
		fUIInRtStatOff(ADR(tyP0934AW.tyMotionStd.tyBtnJogOpen.uiMaskRtStat));
		fUIInRtStatOff(ADR(tyP0934AW.tyMotionStd.tyBtnJogClose.uiMaskRtStat));
		fUIInRtStatOff(ADR(tyP0934AW.tyAW.tyBtnGo.uiMaskRtStat));

	ELSIF tyP0934AW.tyMotionStd.tyBtnMovAbs.bRtCompl = TRUE THEN
		fUIInRtStatOff(ADR(tyP0934AW.tyMotionStd.tyBtnOrigin.uiMaskRtStat));
		fUIInRtStatOff(ADR(tyP0934AW.tyMotionStd.tyBtnMovRel.uiMaskRtStat));
		fUIInRtStatOff(ADR(tyP0934AW.tyMotionStd.tyBtnJogOpen.uiMaskRtStat));
		fUIInRtStatOff(ADR(tyP0934AW.tyMotionStd.tyBtnJogClose.uiMaskRtStat));
		fUIInRtStatOff(ADR(tyP0934AW.tyAW.tyBtnGo.uiMaskRtStat));

	ELSIF tyP0934AW.tyMotionStd.tyBtnMovRel.bRtCompl = TRUE THEN
		fUIInRtStatOff(ADR(tyP0934AW.tyMotionStd.tyBtnOrigin.uiMaskRtStat));
		fUIInRtStatOff(ADR(tyP0934AW.tyMotionStd.tyBtnMovAbs.uiMaskRtStat));
		fUIInRtStatOff(ADR(tyP0934AW.tyMotionStd.tyBtnJogOpen.uiMaskRtStat));
		fUIInRtStatOff(ADR(tyP0934AW.tyMotionStd.tyBtnJogClose.uiMaskRtStat));
		fUIInRtStatOff(ADR(tyP0934AW.tyAW.tyBtnGo.uiMaskRtStat));

	ELSIF tyP0934AW.tyMotionStd.tyBtnJogOpen.bRtCompl = TRUE OR tyP0934AW.tyMotionStd.tyBtnJogOpen.bValue = TRUE THEN
		fUIInRtStatOff(ADR(tyP0934AW.tyMotionStd.tyBtnOrigin.uiMaskRtStat));
		fUIInRtStatOff(ADR(tyP0934AW.tyMotionStd.tyBtnMovAbs.uiMaskRtStat));
		fUIInRtStatOff(ADR(tyP0934AW.tyMotionStd.tyBtnMovRel.uiMaskRtStat));
		fUIInRtStatOff(ADR(tyP0934AW.tyMotionStd.tyBtnJogClose.uiMaskRtStat));
		fUIInRtStatOff(ADR(tyP0934AW.tyAW.tyBtnGo.uiMaskRtStat));

	ELSIF tyP0934AW.tyMotionStd.tyBtnJogClose.bRtCompl = TRUE OR tyP0934AW.tyMotionStd.tyBtnJogClose.bValue = TRUE THEN
		fUIInRtStatOff(ADR(tyP0934AW.tyMotionStd.tyBtnOrigin.uiMaskRtStat));
		fUIInRtStatOff(ADR(tyP0934AW.tyMotionStd.tyBtnMovAbs.uiMaskRtStat));
		fUIInRtStatOff(ADR(tyP0934AW.tyMotionStd.tyBtnMovRel.uiMaskRtStat));
		fUIInRtStatOff(ADR(tyP0934AW.tyMotionStd.tyBtnJogOpen.uiMaskRtStat));
		fUIInRtStatOff(ADR(tyP0934AW.tyAW.tyBtnGo.uiMaskRtStat));

	ELSIF tyP0934AW.tyAW.tyBtnGo.bRtCompl = TRUE THEN
		fUIInRtStatOff(ADR(tyP0934AW.tyMotionStd.tyBtnOrigin.uiMaskRtStat));
		fUIInRtStatOff(ADR(tyP0934AW.tyMotionStd.tyBtnMovAbs.uiMaskRtStat));
		fUIInRtStatOff(ADR(tyP0934AW.tyMotionStd.tyBtnMovRel.uiMaskRtStat));
		fUIInRtStatOff(ADR(tyP0934AW.tyMotionStd.tyBtnJogOpen.uiMaskRtStat));
		fUIInRtStatOff(ADR(tyP0934AW.tyMotionStd.tyBtnJogClose.uiMaskRtStat));

	END_IF

	//Axis Error
	IF tyP0934AW.tyMotionStd.tyBtnPwr.bRtCompl = TRUE THEN
		fUIInRtStatOff(ADR(tyP0934AW.tyMotionStd.tyBtnRst.uiMaskRtStat));
	ELSE
		fUIInRtStatHide(ADR(tyP0934AW.tyMotionStd.tyBtnRst.uiMaskRtStat));
	END_IF

END_ACTION
```

#### Act_OptP0934UpdtDat.st
```iecst
ACTION Act_OptP0934UpdtDat:

	tyP0934AW.tyMotionStd.tyNumCurrPos.diValue			:= p_diAWOpenActualPos;
	tyP0934AW.tyMotionStd.tyNumErrCode.diValue			:= UDINT_TO_DINT(p_udiAWOpenAxisErrID);
	tyP0934AW.tyMotionStd.tyBitmapPwr.usiValueIdx		:= BOOL_TO_USINT(p_bAWOpenPwrOn);
	tyP0934AW.tyMotionStd.tyBitmapRst.usiValueIdx		:= BOOL_TO_USINT(NOT p_bAWOpenAxisErr);
	tyP0934AW.tyMotionStd.tyBitmapOrigin.usiValueIdx	:= BOOL_TO_USINT(p_bAWOpenIsHomed);
	tyP0934AW.tyMotionStd.tyBtnOpenLmtSen.bValue		:= p_bAWOpenOpenSen;
	tyP0934AW.tyMotionStd.tyBtnCloseLmtSen.bValue		:= p_bAWOpenCloseSen;

	//Machine Bitmap
	IF p_bAWOpenIsHomed = TRUE THEN
		IF p_diAWOpenActualPos <= (p_tyNtParamCurr.tyProdRcpWidth.diMax / 2) THEN
			tyP0934AW.tyMotionStd.tyBitmapMc.uiValueIdx 	:= 0;
		ELSE
			tyP0934AW.tyMotionStd.tyBitmapMc.uiValueIdx 	:= 1;
		END_IF
	ELSE
		tyP0934AW.tyMotionStd.tyBitmapMc.uiValueIdx	:= 0;
	END_IF

	IF p_tyNtParamCurr.eProjMag = ULMagDual THEN
		IF p_tyNtParamCurr.bMagAutoVerifyPrep = FALSE THEN
			IF 	tyP0934AW.tyMotionStd.tyBitmapMc.uiValueIdx < 100 THEN
				tyP0934AW.tyMotionStd.tyBitmapMc.uiValueIdx	:= tyP0934AW.tyMotionStd.tyBitmapMc.uiValueIdx + 300;
			END_IF
		ELSE
			IF 	tyP0934AW.tyMotionStd.tyBitmapMc.uiValueIdx < 100 THEN
				tyP0934AW.tyMotionStd.tyBitmapMc.uiValueIdx	:= tyP0934AW.tyMotionStd.tyBitmapMc.uiValueIdx + 300;
			END_IF
		END_IF
	ELSIF p_tyNtParamCurr.eProjMag = ULMagTriple AND p_tyNtParamCurr.bMagAutoVerifyPrep = TRUE AND p_tyNtParamCurr.bProjMotorizedPusherPrep = FALSE THEN
		IF 	tyP0934AW.tyMotionStd.tyBitmapMc.uiValueIdx < 200 THEN
			tyP0934AW.tyMotionStd.tyBitmapMc.uiValueIdx	:= tyP0934AW.tyMotionStd.tyBitmapMc.uiValueIdx + 200;
		END_IF
	ELSIF p_tyNtParamCurr.eProjMag = ULMagTriple AND p_tyNtParamCurr.bMagAutoVerifyPrep = FALSE AND p_tyNtParamCurr.bProjMotorizedPusherPrep = TRUE THEN
		IF 	tyP0934AW.tyMotionStd.tyBitmapMc.uiValueIdx < 400 THEN
			tyP0934AW.tyMotionStd.tyBitmapMc.uiValueIdx	:= tyP0934AW.tyMotionStd.tyBitmapMc.uiValueIdx + 400;
		END_IF
	END_IF

END_ACTION
```

#### Act_OptP0934Keypad.st
```iecst
ACTION Act_OptP0934Keypad:

	IF fUIOutRtStatTPIsOpen(ADR(tyP0934AW.tyAW.tyNumNewWidth.uiRtStat)) = TRUE THEN
		tyProperty.tyKeypad.tyStringTitle.sKeypadTitle		:= tyP0934AW.tyAW.tyNumNewWidth.sKeypadTitle;

	ELSIF fUIOutRtStatTPIsOpen(ADR(tyP0934AW.tyMotionStd.tyNumTargetPos.uiRtStat)) = TRUE THEN
		tyProperty.tyKeypad.tyStringTitle.sKeypadTitle		:= tyP0934AW.tyMotionStd.tyNumTargetPos.sKeypadTitle;

	ELSIF fUIOutRtStatTPIsOpen(ADR(tyP0934AW.tyMotionStd.tyNumStepSize.uiRtStat)) = TRUE THEN
		tyProperty.tyKeypad.tyStringTitle.sKeypadTitle		:= tyP0934AW.tyMotionStd.tyNumStepSize.sKeypadTitle;

	ELSIF fUIOutRtStatTPIsOpen(ADR(tyP0934AW.tyMotionStd.tyNumNomSpd.uiRtStat)) = TRUE THEN
		tyProperty.tyKeypad.tyStringTitle.sKeypadTitle		:= tyP0934AW.tyMotionStd.tyNumNomSpd.sKeypadTitle;

	ELSIF fUIOutRtStatTPIsOpen(ADR(tyP0934AW.tyMotionStd.tyNumSlwSpd.uiRtStat)) = TRUE THEN
		tyProperty.tyKeypad.tyStringTitle.sKeypadTitle		:= tyP0934AW.tyMotionStd.tyNumSlwSpd.sKeypadTitle;

	END_IF

END_ACTION
```

#### Act_OptP0934RstMnl.st
```iecst
ACTION Act_OptP0934RstMnl:

	IF EDGEPOS((bManualMod = FALSE) OR (p_eAWOpenStatus = Error)) THEN

		eAWOpenAct	:= AWActIdle;

		bJogSlow				:= FALSE;
		bJogFast				:= FALSE;
		fbJogSlowToFastDlyTm.IN	:= FALSE;

		tyP0934AW.tyAW.tyBtnGo.bRtCompl					:= FALSE;
		tyP0934AW.tyAW.tyBtnGo.bValue					:= FALSE;
		tyP0934AW.tyAW.tyBtnGo.bRtLk					:= FALSE;
		tyP0934AW.tyAW.tyBtnGo.uiMaskRtStat.0			:= FALSE;

		tyP0934AW.tyMotionStd.tyBtnPwr.bRtCompl				:= FALSE;
		tyP0934AW.tyMotionStd.tyBtnStop.bRtCompl			:= FALSE;
		tyP0934AW.tyMotionStd.tyBtnOrigin.bRtCompl			:= FALSE;
		tyP0934AW.tyMotionStd.tyBtnRst.bRtCompl				:= FALSE;
		tyP0934AW.tyMotionStd.tyBtnMovAbs.bRtCompl			:= FALSE;
		tyP0934AW.tyMotionStd.tyBtnMovRel.bRtCompl			:= FALSE;
		tyP0934AW.tyMotionStd.tyBtnJogOpen.bRtCompl			:= FALSE;
		tyP0934AW.tyMotionStd.tyBtnJogClose.bRtCompl		:= FALSE;

		tyP0934AW.tyMotionStd.tyBtnPwr.bValue				:= FALSE;
		tyP0934AW.tyMotionStd.tyBtnStop.bValue				:= TRUE;
		tyP0934AW.tyMotionStd.tyBtnOrigin.bValue			:= FALSE;
		tyP0934AW.tyMotionStd.tyBtnRst.bValue				:= FALSE;
		tyP0934AW.tyMotionStd.tyBtnMovAbs.bValue			:= FALSE;
		tyP0934AW.tyMotionStd.tyBtnMovRel.bValue			:= FALSE;
		tyP0934AW.tyMotionStd.tyBtnJogOpen.bValue			:= FALSE;
		tyP0934AW.tyMotionStd.tyBtnJogClose.bValue			:= FALSE;

		tyP0934AW.tyMotionStd.tyBtnPwr.bRtLk				:= FALSE;
		tyP0934AW.tyMotionStd.tyBtnStop.bRtLk				:= TRUE;
		tyP0934AW.tyMotionStd.tyBtnOrigin.bRtLk				:= FALSE;
		tyP0934AW.tyMotionStd.tyBtnRst.bRtLk				:= FALSE;
		tyP0934AW.tyMotionStd.tyBtnMovAbs.bRtLk				:= FALSE;
		tyP0934AW.tyMotionStd.tyBtnMovRel.bRtLk				:= FALSE;
		tyP0934AW.tyMotionStd.tyBtnJogOpen.bRtLk			:= FALSE;
		tyP0934AW.tyMotionStd.tyBtnJogClose.bRtLk			:= FALSE;

		tyP0934AW.tyMotionStd.tyBtnPwr.uiMaskRtStat			:= TRUE;
		tyP0934AW.tyMotionStd.tyBtnOrigin.uiMaskRtStat		:= FALSE;
		tyP0934AW.tyMotionStd.tyBtnRst.uiMaskRtStat			:= TRUE;
		tyP0934AW.tyMotionStd.tyBtnMovAbs.uiMaskRtStat		:= FALSE;
		tyP0934AW.tyMotionStd.tyBtnMovRel.uiMaskRtStat		:= FALSE;
		tyP0934AW.tyMotionStd.tyBtnJogOpen.uiMaskRtStat		:= FALSE;
		tyP0934AW.tyMotionStd.tyBtnJogClose.uiMaskRtStat	:= FALSE;

	END_IF

	eInShutterAct	:= PneuActIdle;
	eOutShutterAct	:= PneuActIdle;

	tyP0934AW.tyInOutletShutterFB.tyBtnClose.bRtCompl	:= FALSE;
	tyP0934AW.tyInOutletShutterFB.tyBtnClose.bValue	:= FALSE;
	tyP0934AW.tyInOutletShutterFB.tyBtnOpen.bRtCompl	:= FALSE;
	tyP0934AW.tyInOutletShutterFB.tyBtnOpen.bValue	:= FALSE;

END_ACTION
```

#### Act_EntP0935Disp.st
```iecst
ACTION Act_EntP0935Disp:

	//Access Address
	p_tyC0001MotionStd ACCESS ADR(tyP0935Lifter.tyMotionStd);

	p_tyC0002FullMask ACCESS ADR(tyP0935Lifter.tyFullMaskHide);

	p_tyC0004Navi ACCESS ADR(tyP0935Lifter.tyNaviBack);

	p_tyC0005Main ACCESS ADR(tyCommon.tyMain);

	p_tyC0007Notif ACCESS ADR(tyCommon.tyNotif);

	p_tyC0008MsgBox ACCESS ADR(tyP0935Lifter.tyMsgBoxHide);

	p_tyC0009Info ACCESS ADR(tyCommon.tyInfo);

	p_tyP0935Lifter ACCESS ADR(tyP0935Lifter.tyLifter);

	p_tyP0935InOutletShutterFB ACCESS ADR(tyP0935Lifter.tyInOutletShutterFB);

	//Display
	tyP0935Lifter.tyMotionStd.tyBtnPwr.bValue	:= p_bLifterBtmPwrOn;

	tyP0935Lifter.tyLifter.tyNumNewSlt.diValueMax	:= p_tyMagRcpCurrRcp.diTtlSlt;

END_ACTION
```

#### Act_OptP0935Navi.st
```iecst
ACTION Act_OptP0935Navi:

	IF tyP0935Lifter.tyNaviBack.tyBtnBack.bRtCompl = TRUE THEN
		tyP0935Lifter.tyNaviBack.tyBtnBack.bRtCompl	:= FALSE;
		tyP0935Lifter.tyNaviBack.tyBtnBack.bValue	:= FALSE;

		eChgPage	:= UIP0920MtrNPneuCtrl;

	END_IF

END_ACTION
```

#### Act_OptP0935FullMask.st
```iecst
ACTION Act_OptP0935FullMask:

	IF eCurrPage = UIP0935Lifter THEN

		IF p_tyDI.bEStopSig = FALSE THEN
			p_tyC0002FullMask ACCESS ADR(tyP0935Lifter.tyFullMaskEStop);

		ELSIF p_tyDI.bCoverSWSig = FALSE THEN
			p_tyC0002FullMask ACCESS ADR(tyP0935Lifter.tyFullMaskCWSig);

		ELSIF p_tyDI.bSafetyRlySig = FALSE THEN
			p_tyC0002FullMask ACCESS ADR(tyP0935Lifter.tyFullMaskSafetyRly);

		ELSIF p_tyDI.bPusherExtRS = TRUE THEN
			p_tyC0002FullMask ACCESS ADR(tyP0935Lifter.tyFullMaskPshrInterrupt);
		ELSIF p_tyDI.bPusherRetRS = FALSE AND p_tyDI.bPusherRetSlwSen = FALSE  THEN
			p_tyC0002FullMask ACCESS ADR(tyP0936Trav.tyFullMaskPshrNotRetInterrupt);
		ELSIF (p_tyNtParamCurr.bProjInletShutPrep AND p_tyDI.bInShutterCloseRS = FALSE) AND NOT(bBypassShutForCalib) THEN
			p_tyC0002FullMask ACCESS ADR(tyP0935Lifter.tyFullMaskInShutOpnInterrupt);

		ELSIF ((p_tyDI.bOutShutterCloseRS = FALSE AND p_tyNtParamCurr.bProjOutletShutPrep) OR (p_tyDI.bOutShutterCloseRS2 = FALSE AND p_tyNtParamCurr.bProjOutletShut2Prep )OR (p_tyDI.bOutShutterCloseRS3 = FALSE AND p_tyNtParamCurr.bProjOutletShut3Prep)) AND NOT(bBypassShutForCalib) THEN
			IF p_tyNtParamCurr.bCurtainSenPrep THEN
				IF (p_tyDI.bOutShutterCloseRS = FALSE AND p_tyNtParamCurr.bProjOutletShutPrep) OR (p_tyDI.bOutShutterCloseRS2 = FALSE AND p_tyNtParamCurr.bProjOutletShut2Prep)OR (p_tyDI.bOutShutterCloseRS3 = FALSE AND p_tyNtParamCurr.bProjOutletShut3Prep )THEN
					p_tyC0002FullMask ACCESS ADR(tyP0935Lifter.tyFullMaskOutShutOpnInterrupt);
				END_IF
			ELSE
				IF p_tyDI.bOutShutterCloseRS = FALSE THEN
					p_tyC0002FullMask ACCESS ADR(tyP0935Lifter.tyFullMaskOutShutOpnInterrupt);
				END_IF
			END_IF

		ELSIF p_tyDI.bConvLftSen THEN
			p_tyC0002FullMask ACCESS ADR(tyP0935Lifter.tyFullMaskLftSenInterrupt);

		ELSIF p_tyDI.bConvClrSen THEN
			p_tyC0002FullMask ACCESS ADR(tyP0935Lifter.tyFullMaskClrSenInterrupt);

//		ELSIF p_tyDI.bLifterSafetyLmtSW1 = FALSE OR p_tyDI.bLifterSafetyLmtSW2 = FALSE THEN
//			p_tyC0002FullMask ACCESS ADR(tyP0935Lifter.tyFullMaskSafetyLmtSW);
//			kyumin request to hide
		ELSIF p_tyDI.bLifterTimingBeltSen = FALSE THEN
			p_tyC0002FullMask ACCESS ADR(tyP0935Lifter.tyFullMaskTimingBelt);

//		ELSIF p_tyNtParamCurr.tyDISettings.diMag1FixedClampRS <> 0 AND p_tyDI.bMag1FixedClampRS = FALSE
//			AND p_tyDI.bMagPresentSen1 THEN
//			p_tyC0002FullMask ACCESS ADR(tyP0935Lifter.tyFullMaskMagClmpInt);
		ELSE
			p_tyC0002FullMask ACCESS ADR(tyP0935Lifter.tyFullMaskHide);

		END_IF

	END_IF

END_ACTION
```

#### Act_OptP0935FBCtrl.st
```iecst
ACTION Act_OptP0935FBCtrl:

	fbJogSlowToFastDlyTm.PT	:= T#2s;
	fbJogSlowToFastDlyTm;
	fbLmtRstTm;

	//Lifter Safety Sensor Interruption
	IF EDGENEG(p_tyDI.bLifterSafetyLmtSW1 AND p_tyDI.bLifterSafetyLmtSW2 AND p_tyDI.bLifterTimingBeltSen) THEN
		tyP0935Lifter.tyMotionStd.tyBtnStop.bRtCompl	:= TRUE;
	END_IF

//	IF EDGEPOS((p_udiLifterBtmAxisErrID = 21570 OR p_udiLifterBtmAxisErrID = 21571)
	IF EDGEPOS((p_bLifterBtmFwdLmtSen OR p_bLifterBtmRevLmtSen OR p_udiLifterBtmAxisErrID = 21570 OR p_udiLifterBtmAxisErrID = 21571)
		AND tyP0935Lifter.tyMotionStd.tyBtnJogDown.bValue = FALSE
		AND tyP0935Lifter.tyMotionStd.tyBtnJogUp.bValue = FALSE)
	THEN
		fbLmtRstTm.IN				:= TRUE;
	END_IF

	IF fbLmtRstTm.Q = TRUE THEN
		tyP0935Lifter.tyMotionStd.tyBtnRst.bRtCompl		:= TRUE;
	END_IF

	IF (tyP0935Lifter.tyMotionStd.tyBtnJogUp.bValue = FALSE AND tyP0935Lifter.tyMotionStd.tyBtnJogDown.bValue = FALSE) AND (p_bLifterBtmJogging = TRUE) THEN
		bJogStopLifter	:= TRUE;
	END_IF

	IF tyP0935Lifter.tyMotionStd.tyBtnStop.bRtCompl = TRUE THEN
		eLifterBtmAct		:= LifterActStop;

		IF p_eLifterBtmStat = LifterActStop AND p_eLifterBtmStatus = Done THEN
			eLifterBtmAct	:= LifterActIdle;

			tyP0935Lifter.tyMotionStd.tyBtnStop.bRtCompl			:= FALSE;
			tyP0935Lifter.tyMotionStd.tyBtnJogDown.bRtCompl			:= FALSE;
			tyP0935Lifter.tyMotionStd.tyBtnJogUp.bRtCompl			:= FALSE;
			tyP0935Lifter.tyMotionStd.tyBtnOrigin.bRtCompl			:= FALSE;
			tyP0935Lifter.tyMotionStd.tyBtnMovAbs.bRtCompl			:= FALSE;
			tyP0935Lifter.tyMotionStd.tyBtnMovRel.bRtCompl			:= FALSE;
			tyP0935Lifter.tyLifter.tyBtnGo.bRtCompl					:= FALSE;
			tyP0935Lifter.tyLifter.tyBtnNxtSlt.bRtCompl				:= FALSE;
			tyP0935Lifter.tyLifter.tyBtnPrevSlt.bRtCompl			:= FALSE;
			tyP0935Lifter.tyLifter.tyBtnGoLaneA.bRtCompl			:= FALSE;
			tyP0935Lifter.tyLifter.tyBtnGoLaneB.bRtCompl			:= FALSE;
			tyP0935Lifter.tyLifter.tyBtnGoLaneD_G.bRtCompl			:= FALSE;
			tyP0935Lifter.tyLifter.tyBtnGoLaneE_H.bRtCompl			:= FALSE;

			tyP0935Lifter.tyMotionStd.tyBtnStop.bValue				:= TRUE;
			tyP0935Lifter.tyMotionStd.tyBtnJogDown.bValue			:= FALSE;
			tyP0935Lifter.tyMotionStd.tyBtnJogUp.bValue				:= FALSE;
			tyP0935Lifter.tyMotionStd.tyBtnOrigin.bValue			:= FALSE;
			tyP0935Lifter.tyMotionStd.tyBtnMovAbs.bValue			:= FALSE;
			tyP0935Lifter.tyMotionStd.tyBtnMovRel.bValue			:= FALSE;
			tyP0935Lifter.tyLifter.tyBtnGo.bValue					:= FALSE;
			tyP0935Lifter.tyLifter.tyBtnNxtSlt.bValue				:= FALSE;
			tyP0935Lifter.tyLifter.tyBtnPrevSlt.bValue				:= FALSE;
			tyP0935Lifter.tyLifter.tyBtnGoLaneA.bValue				:= FALSE;
			tyP0935Lifter.tyLifter.tyBtnGoLaneB.bValue				:= FALSE;
			tyP0935Lifter.tyLifter.tyBtnGoLaneD_G.bValue			:= FALSE;
			tyP0935Lifter.tyLifter.tyBtnGoLaneE_H.bValue			:= FALSE;

			tyP0935Lifter.tyMotionStd.tyBtnStop.bRtLk				:= TRUE;
			tyP0935Lifter.tyMotionStd.tyBtnJogDown.bRtLk			:= FALSE;
			tyP0935Lifter.tyMotionStd.tyBtnJogUp.bRtLk				:= FALSE;
			tyP0935Lifter.tyMotionStd.tyBtnOrigin.bRtLk				:= FALSE;
			tyP0935Lifter.tyMotionStd.tyBtnMovAbs.bRtLk				:= FALSE;
			tyP0935Lifter.tyMotionStd.tyBtnMovRel.bRtLk				:= FALSE;
			tyP0935Lifter.tyLifter.tyBtnGo.bRtLk					:= FALSE;
			tyP0935Lifter.tyLifter.tyBtnNxtSlt.bRtLk				:= FALSE;
			tyP0935Lifter.tyLifter.tyBtnPrevSlt.bRtLk				:= FALSE;
			tyP0935Lifter.tyLifter.tyBtnGoLaneA.bRtLk				:= FALSE;
			tyP0935Lifter.tyLifter.tyBtnGoLaneB.bRtLk				:= FALSE;
			tyP0935Lifter.tyLifter.tyBtnGoLaneD_G.bRtLk				:= FALSE;
			tyP0935Lifter.tyLifter.tyBtnGoLaneE_H.bRtLk				:= FALSE;

		END_IF

	ELSIF (tyP0935Lifter.tyMotionStd.tyBtnJogDown.bRtCompl = TRUE) OR (tyP0935Lifter.tyMotionStd.tyBtnJogUp.bRtCompl = TRUE) OR (bJogStopLifter = TRUE) THEN
		bJogSlow					:= FALSE;
		bJogFast					:= FALSE;
		fbJogSlowToFastDlyTm.IN		:= FALSE;

		eLifterBtmAct		:= LifterActJogStop;

		IF p_eLifterBtmStat = LifterActJogStop AND p_eLifterBtmStatus = Done THEN
			eLifterBtmAct		:= LifterActIdle;

			bJogStopLifter	:= FALSE;

			tyP0935Lifter.tyMotionStd.tyBtnStop.bRtCompl			:= FALSE;
			tyP0935Lifter.tyMotionStd.tyBtnJogDown.bRtCompl			:= FALSE;
			tyP0935Lifter.tyMotionStd.tyBtnJogUp.bRtCompl			:= FALSE;
			tyP0935Lifter.tyMotionStd.tyBtnOrigin.bRtCompl			:= FALSE;
			tyP0935Lifter.tyMotionStd.tyBtnMovAbs.bRtCompl			:= FALSE;
			tyP0935Lifter.tyMotionStd.tyBtnMovRel.bRtCompl			:= FALSE;
			tyP0935Lifter.tyLifter.tyBtnGo.bRtCompl					:= FALSE;
			tyP0935Lifter.tyLifter.tyBtnNxtSlt.bRtCompl				:= FALSE;
			tyP0935Lifter.tyLifter.tyBtnPrevSlt.bRtCompl			:= FALSE;

			tyP0935Lifter.tyMotionStd.tyBtnStop.bValue				:= TRUE;
			tyP0935Lifter.tyMotionStd.tyBtnJogDown.bValue			:= FALSE;
			tyP0935Lifter.tyMotionStd.tyBtnJogUp.bValue				:= FALSE;
			tyP0935Lifter.tyMotionStd.tyBtnOrigin.bValue			:= FALSE;
			tyP0935Lifter.tyMotionStd.tyBtnMovAbs.bValue			:= FALSE;
			tyP0935Lifter.tyMotionStd.tyBtnMovRel.bValue			:= FALSE;
			tyP0935Lifter.tyLifter.tyBtnGo.bValue					:= FALSE;
			tyP0935Lifter.tyLifter.tyBtnNxtSlt.bValue				:= FALSE;
			tyP0935Lifter.tyLifter.tyBtnPrevSlt.bValue				:= FALSE;

			tyP0935Lifter.tyMotionStd.tyBtnStop.bRtLk				:= TRUE;
			tyP0935Lifter.tyMotionStd.tyBtnJogDown.bRtLk			:= FALSE;
			tyP0935Lifter.tyMotionStd.tyBtnJogUp.bRtLk				:= FALSE;
			tyP0935Lifter.tyMotionStd.tyBtnOrigin.bRtLk				:= FALSE;
			tyP0935Lifter.tyMotionStd.tyBtnMovAbs.bRtLk				:= FALSE;
			tyP0935Lifter.tyMotionStd.tyBtnMovRel.bRtLk				:= FALSE;
			tyP0935Lifter.tyLifter.tyBtnGo.bRtLk					:= FALSE;
			tyP0935Lifter.tyLifter.tyBtnNxtSlt.bRtLk				:= FALSE;
			tyP0935Lifter.tyLifter.tyBtnPrevSlt.bRtLk				:= FALSE;

		END_IF

	ELSIF tyP0935Lifter.tyMotionStd.tyBtnPwr.bRtCompl = TRUE THEN
		tyP0935Lifter.tyMotionStd.tyBtnPwr.bRtLk					:= TRUE;

		IF tyP0935Lifter.tyMotionStd.tyBtnPwr.bValue = TRUE THEN
			eLifterBtmAct		:= LifterActPwrOn;

			IF p_eLifterBtmStat = LifterActPwrOn AND p_eLifterBtmStatus = Done THEN
				eLifterBtmAct	:= LifterActIdle;

				tyP0935Lifter.tyMotionStd.tyBtnPwr.bRtCompl		:= FALSE;
				tyP0935Lifter.tyMotionStd.tyBtnPwr.bRtLk		:= FALSE;
			END_IF
		ELSE
			eLifterBtmAct		:= LifterActPwrOff;

			IF p_eLifterBtmStat = LifterActPwrOff AND p_eLifterBtmStatus = Done THEN
				eLifterBtmAct	:= LifterActIdle;

				tyP0935Lifter.tyMotionStd.tyBtnPwr.bRtCompl		:= FALSE;
				tyP0935Lifter.tyMotionStd.tyBtnPwr.bRtLk		:= FALSE;
			END_IF
		END_IF

	ELSIF tyP0935Lifter.tyMotionStd.tyBtnOrigin.bRtCompl = TRUE THEN
		tyP0935Lifter.tyMotionStd.tyBtnOrigin.bValue				:= TRUE;
		tyP0935Lifter.tyMotionStd.tyBtnStop.bValue					:= FALSE;

		tyP0935Lifter.tyMotionStd.tyBtnOrigin.bRtLk					:= TRUE;
		tyP0935Lifter.tyMotionStd.tyBtnStop.bRtLk					:= FALSE;

		eLifterBtmAct		:= LifterActHoming;

		IF p_eLifterBtmStat = LifterActHoming AND p_eLifterBtmStatus = Done THEN
			eLifterBtmAct	:= LifterActIdle;

			tyP0935Lifter.tyMotionStd.tyBtnOrigin.bRtCompl		:= FALSE;
			tyP0935Lifter.tyMotionStd.tyBtnOrigin.bValue		:= FALSE;
			tyP0935Lifter.tyMotionStd.tyBtnStop.bValue			:= TRUE;

			tyP0935Lifter.tyMotionStd.tyBtnOrigin.bRtLk			:= FALSE;
			tyP0935Lifter.tyMotionStd.tyBtnStop.bRtLk			:= TRUE;

		END_IF

	ELSIF tyP0935Lifter.tyMotionStd.tyBtnRst.bRtCompl = TRUE THEN
		tyP0935Lifter.tyMotionStd.tyBtnRst.bValue				:= TRUE;
		tyP0935Lifter.tyMotionStd.tyBtnRst.bRtLk				:= TRUE;

		eLifterBtmAct		:= LifterActRstAxisErr;

		IF p_eLifterBtmStat = LifterActRstAxisErr AND p_eLifterBtmStatus = Done THEN
			eLifterBtmAct	:= LifterActIdle;

			tyP0935Lifter.tyMotionStd.tyBtnRst.bRtCompl			:= FALSE;
			tyP0935Lifter.tyMotionStd.tyBtnRst.bValue			:= FALSE;
			tyP0935Lifter.tyMotionStd.tyBtnRst.bRtLk			:= FALSE;

			fbLmtRstTm.IN			:= FALSE;
		END_IF

	ELSIF tyP0935Lifter.tyLifter.tyBtnGo.bRtCompl = TRUE THEN
		tyP0935Lifter.tyLifter.tyBtnGo.bValue				:= TRUE;
		tyP0935Lifter.tyMotionStd.tyBtnStop.bValue			:= FALSE;

		tyP0935Lifter.tyLifter.tyBtnGo.bRtLk				:= TRUE;
		tyP0935Lifter.tyMotionStd.tyBtnStop.bRtLk			:= FALSE;

		(*diMnlLifterMag1GoSlt	:= tyP0935Lifter.tyLifter.tyNumNewSlt.diValue;*)
		diMnlLifterNomSpd		:= tyP0935Lifter.tyMotionStd.tyNumNomSpd.diValue;

		CASE tyP0935Lifter.tyLifter.tyNumMagPos.diValue OF
			1:
				eLifterBtmAct	:= LifterActGoASltPos;
				diMnlLifterMag1GoSlt	:= tyP0935Lifter.tyLifter.tyNumNewSlt.diValue;

			2:
				eLifterBtmAct	:= LifterActGoBSltPos;
				diMnlLifterMag2GoSlt	:= tyP0935Lifter.tyLifter.tyNumNewSlt.diValue;

			3:
				eLifterBtmAct	:= LifterActGoCSltPos;
				diMnlLifterMag3GoSlt	:= tyP0935Lifter.tyLifter.tyNumNewSlt.diValue;

			4:
				eLifterBtmAct	:= LifterActGoDSltPos;
				diMnlLifterMag3GoSlt	:= tyP0935Lifter.tyLifter.tyNumNewSlt.diValue;
		END_CASE

		IF (p_eLifterBtmStat = LifterActGoASltPos
			OR p_eLifterBtmStat = LifterActGoBSltPos
			OR p_eLifterBtmStat = LifterActGoCSltPos
			OR p_eLifterBtmStat = LifterActGoDSltPos)
			AND p_eLifterBtmStatus = Done THEN
			eLifterBtmAct	:= LifterActIdle;

			tyP0935Lifter.tyLifter.tyBtnGo.bRtCompl				:= FALSE;
			tyP0935Lifter.tyLifter.tyBtnGo.bValue				:= FALSE;
			tyP0935Lifter.tyMotionStd.tyBtnStop.bValue			:= TRUE;

			tyP0935Lifter.tyLifter.tyBtnGo.bRtLk				:= FALSE;
			tyP0935Lifter.tyMotionStd.tyBtnStop.bRtLk			:= TRUE;
		END_IF

	ELSIF tyP0935Lifter.tyLifter.tyBtnNxtSlt.bRtCompl = TRUE THEN
		tyP0935Lifter.tyLifter.tyBtnNxtSlt.bValue				:= TRUE;
		tyP0935Lifter.tyMotionStd.tyBtnStop.bValue				:= FALSE;

		tyP0935Lifter.tyLifter.tyBtnNxtSlt.bRtLk				:= TRUE;
		tyP0935Lifter.tyMotionStd.tyBtnStop.bRtLk				:= FALSE;

		(*diMnlLifterMag1GoSlt	:= tyP0935Lifter.tyLifter.tyNumNewSlt.diValue;*)
		diMnlLifterNomSpd		:= tyP0935Lifter.tyMotionStd.tyNumNomSpd.diValue;

		CASE tyP0935Lifter.tyLifter.tyNumMagPos.diValue OF
			1:
				eLifterBtmAct	:= LifterActGoNxtASltPos;
				diMnlLifterMag1GoSlt	:= tyP0935Lifter.tyLifter.tyNumNewSlt.diValue;
			2:
				eLifterBtmAct	:= LifterActGoNxtBSltPos;
				diMnlLifterMag2GoSlt	:= tyP0935Lifter.tyLifter.tyNumNewSlt.diValue;
			3:
				eLifterBtmAct	:= LifterActGoNxtCSltPos;
				diMnlLifterMag3GoSlt	:= tyP0935Lifter.tyLifter.tyNumNewSlt.diValue;
			4:
				eLifterBtmAct	:= LifterActGoNxtDSltPos;
		//		diMnlLifterMag4GoSlt	:= tyP0935Lifter.tyLifter.tyNumNewSlt.diValue;

		END_CASE

		IF (p_eLifterBtmStat = LifterActGoNxtASltPos
			OR p_eLifterBtmStat = LifterActGoNxtBSltPos
			OR p_eLifterBtmStat = LifterActGoNxtCSltPos
			OR p_eLifterBtmStat = LifterActGoNxtDSltPos)
			AND p_eLifterBtmStatus = Done THEN
			eLifterBtmAct	:= LifterActIdle;

			tyP0935Lifter.tyLifter.tyBtnNxtSlt.bRtCompl				:= FALSE;
			tyP0935Lifter.tyLifter.tyBtnNxtSlt.bValue				:= FALSE;
			tyP0935Lifter.tyMotionStd.tyBtnStop.bValue				:= TRUE;

			tyP0935Lifter.tyLifter.tyBtnNxtSlt.bRtLk				:= FALSE;
			tyP0935Lifter.tyMotionStd.tyBtnStop.bRtLk				:= TRUE;
		END_IF

	ELSIF tyP0935Lifter.tyLifter.tyBtnPrevSlt.bRtCompl = TRUE THEN
		tyP0935Lifter.tyLifter.tyBtnPrevSlt.bValue				:= TRUE;
		tyP0935Lifter.tyMotionStd.tyBtnStop.bValue				:= FALSE;

		tyP0935Lifter.tyLifter.tyBtnPrevSlt.bRtLk				:= TRUE;
		tyP0935Lifter.tyMotionStd.tyBtnStop.bRtLk				:= FALSE;

	//	diMnlLifterMag1GoSlt	:= tyP0935Lifter.tyLifter.tyNumNewSlt.diValue;
		diMnlLifterNomSpd		:= tyP0935Lifter.tyMotionStd.tyNumNomSpd.diValue;

		CASE tyP0935Lifter.tyLifter.tyNumMagPos.diValue OF

			1:
				eLifterBtmAct	:= LifterActGoPrevASltPos;
				diMnlLifterMag1GoSlt	:= tyP0935Lifter.tyLifter.tyNumNewSlt.diValue;

			2:
				eLifterBtmAct	:= LifterActGoPrevBSltPos;
				diMnlLifterMag2GoSlt	:= tyP0935Lifter.tyLifter.tyNumNewSlt.diValue;

			3:
				eLifterBtmAct	:= LifterActGoPrevCSltPos;
				diMnlLifterMag3GoSlt	:= tyP0935Lifter.tyLifter.tyNumNewSlt.diValue;

			4:
				eLifterBtmAct	:= LifterActGoPrevDSltPos;
		//		diMnlLifterMag4GoSlt	:= tyP0935Lifter.tyLifter.tyNumNewSlt.diValue;

		END_CASE

		IF (p_eLifterBtmStat = LifterActGoPrevASltPos
			OR p_eLifterBtmStat = LifterActGoPrevBSltPos
			OR p_eLifterBtmStat = LifterActGoPrevCSltPos
			OR p_eLifterBtmStat = LifterActGoPrevDSltPos)
			AND p_eLifterBtmStatus = Done THEN
			eLifterBtmAct	:= LifterActIdle;

			tyP0935Lifter.tyLifter.tyBtnPrevSlt.bRtCompl				:= FALSE;
			tyP0935Lifter.tyLifter.tyBtnPrevSlt.bValue					:= FALSE;
			tyP0935Lifter.tyMotionStd.tyBtnStop.bValue					:= TRUE;

			tyP0935Lifter.tyLifter.tyBtnPrevSlt.bRtLk					:= FALSE;
			tyP0935Lifter.tyMotionStd.tyBtnStop.bRtLk					:= TRUE;
		END_IF

	ELSIF tyP0935Lifter.tyLifter.tyBtnGoLaneA.bRtCompl = TRUE THEN
		tyP0935Lifter.tyLifter.tyBtnGoLaneA.bValue	:= TRUE;
		tyP0935Lifter.tyMotionStd.tyBtnStop.bValue	:= FALSE;

		tyP0935Lifter.tyLifter.tyBtnGoLaneA.bRtLk	:= TRUE;
		tyP0935Lifter.tyMotionStd.tyBtnStop.bRtLk	:= FALSE;

		diMnlLifterNomSpd	:= tyP0935Lifter.tyMotionStd.tyNumNomSpd.diValue;

		eLifterBtmAct	:= LifterActGoAPos;

		IF p_eLifterBtmStat = LifterActGoAPos AND p_eLifterBtmStatus = Done THEN
			eLifterBtmAct	:= LifterActIdle;

			tyP0935Lifter.tyLifter.tyBtnGoLaneA.bRtCompl	:= FALSE;

			tyP0935Lifter.tyLifter.tyBtnGoLaneA.bValue	:= FALSE;
			tyP0935Lifter.tyMotionStd.tyBtnStop.bValue	:= TRUE;

			tyP0935Lifter.tyLifter.tyBtnGoLaneA.bRtLk	:= FALSE;
			tyP0935Lifter.tyMotionStd.tyBtnStop.bRtLk	:= TRUE;
		END_IF

	ELSIF tyP0935Lifter.tyLifter.tyBtnGoLaneB.bRtCompl = TRUE THEN
		tyP0935Lifter.tyLifter.tyBtnGoLaneB.bValue	:= TRUE;
		tyP0935Lifter.tyMotionStd.tyBtnStop.bValue	:= FALSE;

		tyP0935Lifter.tyLifter.tyBtnGoLaneB.bRtLk	:= TRUE;
		tyP0935Lifter.tyMotionStd.tyBtnStop.bRtLk	:= FALSE;

		diMnlLifterNomSpd	:= tyP0935Lifter.tyMotionStd.tyNumNomSpd.diValue;

		eLifterBtmAct	:= LifterActGoBPos;

		IF p_eLifterBtmStat = LifterActGoBPos AND p_eLifterBtmStatus = Done THEN
			eLifterBtmAct	:= LifterActIdle;

			tyP0935Lifter.tyLifter.tyBtnGoLaneB.bRtCompl	:= FALSE;

			tyP0935Lifter.tyLifter.tyBtnGoLaneB.bValue	:= FALSE;
			tyP0935Lifter.tyMotionStd.tyBtnStop.bValue	:= TRUE;

			tyP0935Lifter.tyLifter.tyBtnGoLaneB.bRtLk	:= FALSE;
			tyP0935Lifter.tyMotionStd.tyBtnStop.bRtLk	:= TRUE;
		END_IF

	ELSIF tyP0935Lifter.tyLifter.tyBtnGoLaneD_G.bRtCompl = TRUE THEN
		tyP0935Lifter.tyLifter.tyBtnGoLaneD_G.bValue	:= TRUE;
		tyP0935Lifter.tyMotionStd.tyBtnStop.bValue	:= FALSE;

		tyP0935Lifter.tyLifter.tyBtnGoLaneD_G.bRtLk	:= TRUE;
		tyP0935Lifter.tyMotionStd.tyBtnStop.bRtLk	:= FALSE;

		diMnlLifterNomSpd	:= tyP0935Lifter.tyMotionStd.tyNumNomSpd.diValue;

		eLifterBtmAct	:= LifterActGoDPos;

		IF p_eLifterBtmStat = LifterActGoDPos AND p_eLifterBtmStatus = Done THEN
			eLifterBtmAct	:= LifterActIdle;

			tyP0935Lifter.tyLifter.tyBtnGoLaneD_G.bRtCompl	:= FALSE;

			tyP0935Lifter.tyLifter.tyBtnGoLaneD_G.bValue	:= FALSE;
			tyP0935Lifter.tyMotionStd.tyBtnStop.bValue	:= TRUE;

			tyP0935Lifter.tyLifter.tyBtnGoLaneD_G.bRtLk	:= FALSE;
			tyP0935Lifter.tyMotionStd.tyBtnStop.bRtLk	:= TRUE;
		END_IF

	ELSIF tyP0935Lifter.tyLifter.tyBtnGoLaneE_H.bRtCompl = TRUE THEN
		tyP0935Lifter.tyLifter.tyBtnGoLaneE_H.bValue	:= TRUE;
		tyP0935Lifter.tyMotionStd.tyBtnStop.bValue	:= FALSE;

		tyP0935Lifter.tyLifter.tyBtnGoLaneE_H.bRtLk	:= TRUE;
		tyP0935Lifter.tyMotionStd.tyBtnStop.bRtLk	:= FALSE;

		diMnlLifterNomSpd	:= tyP0935Lifter.tyMotionStd.tyNumNomSpd.diValue;

		eLifterBtmAct	:= LifterActGoEPos;

		IF p_eLifterBtmStat = LifterActGoEPos AND p_eLifterBtmStatus = Done THEN
			eLifterBtmAct	:= LifterActIdle;

			tyP0935Lifter.tyLifter.tyBtnGoLaneE_H.bRtCompl	:= FALSE;

			tyP0935Lifter.tyLifter.tyBtnGoLaneE_H.bValue	:= FALSE;
			tyP0935Lifter.tyMotionStd.tyBtnStop.bValue	:= TRUE;

			tyP0935Lifter.tyLifter.tyBtnGoLaneE_H.bRtLk	:= FALSE;
			tyP0935Lifter.tyMotionStd.tyBtnStop.bRtLk	:= TRUE;
		END_IF

	ELSIF tyP0935Lifter.tyMotionStd.tyBtnMovAbs.bRtCompl = TRUE THEN

		tyP0935Lifter.tyMotionStd.tyBtnMovAbs.bValue				:= TRUE;
		tyP0935Lifter.tyMotionStd.tyBtnStop.bValue					:= FALSE;

		tyP0935Lifter.tyMotionStd.tyBtnMovAbs.bRtLk					:= TRUE;
		tyP0935Lifter.tyMotionStd.tyBtnStop.bRtLk					:= FALSE;

		diMnlLifterTargetPos	:= tyP0935Lifter.tyMotionStd.tyNumTargetPos.diValue;
		diMnlLifterNomSpd		:= tyP0935Lifter.tyMotionStd.tyNumNomSpd.diValue;

		eLifterBtmAct			:= LifterActMovAbs;

		IF p_eLifterBtmStat = LifterActMovAbs AND p_eLifterBtmStatus = Done THEN
			eLifterBtmAct	:= LifterActIdle;

			tyP0935Lifter.tyMotionStd.tyBtnMovAbs.bRtCompl		:= FALSE;
			tyP0935Lifter.tyMotionStd.tyBtnMovAbs.bValue		:= FALSE;
			tyP0935Lifter.tyMotionStd.tyBtnStop.bValue			:= TRUE;

			tyP0935Lifter.tyMotionStd.tyBtnMovAbs.bRtLk			:= FALSE;
			tyP0935Lifter.tyMotionStd.tyBtnStop.bRtLk			:= TRUE;
		END_IF

	ELSIF tyP0935Lifter.tyMotionStd.tyBtnMovRel.bRtCompl = TRUE THEN
		tyP0935Lifter.tyMotionStd.tyBtnMovRel.bValue			:= TRUE;
		tyP0935Lifter.tyMotionStd.tyBtnStop.bValue				:= FALSE;

		tyP0935Lifter.tyMotionStd.tyBtnMovRel.bRtLk				:= TRUE;
		tyP0935Lifter.tyMotionStd.tyBtnStop.bRtLk				:= FALSE;

		diMnlLifterStepSize		:= tyP0935Lifter.tyMotionStd.tyNumStepSize.diValue;
		diMnlLifterNomSpd		:= tyP0935Lifter.tyMotionStd.tyNumNomSpd.diValue;

		eLifterBtmAct		:= LifterActMovRel;

		IF p_eLifterBtmStat = LifterActMovRel AND p_eLifterBtmStatus = Done THEN
			eLifterBtmAct	:= LifterActIdle;

			tyP0935Lifter.tyMotionStd.tyBtnMovRel.bRtCompl		:= FALSE;
			tyP0935Lifter.tyMotionStd.tyBtnMovRel.bValue		:= FALSE;
			tyP0935Lifter.tyMotionStd.tyBtnStop.bValue			:= TRUE;

			tyP0935Lifter.tyMotionStd.tyBtnMovRel.bRtLk			:= FALSE;
			tyP0935Lifter.tyMotionStd.tyBtnStop.bRtLk			:= TRUE;

		END_IF

	ELSIF (tyP0935Lifter.tyMotionStd.tyBtnJogDown.bValue = TRUE) AND (fbJogSlowToFastDlyTm.Q = FALSE) AND (bJogSlow = FALSE) THEN
		tyP0935Lifter.tyMotionStd.tyBtnStop.bValue				:= FALSE;
		tyP0935Lifter.tyMotionStd.tyBtnStop.bRtLk				:= FALSE;

		fbJogSlowToFastDlyTm.IN		:= TRUE;

		diMnlLifterJogSpd	:= tyP0935Lifter.tyMotionStd.tyNumSlwSpd.diValue;

		eLifterBtmAct		:= LifterActJogDown;

		IF p_eLifterBtmStat = LifterActJogDown AND p_eLifterBtmStatus = Done THEN

			eLifterBtmAct	:= LifterActIdle;
			bJogSlow				:= TRUE;

		ELSIF p_eLifterBtmStatus = Error THEN

			fbJogSlowToFastDlyTm.IN	:= FALSE;
			bJogSlow				:= TRUE;

		END_IF

	ELSIF (tyP0935Lifter.tyMotionStd.tyBtnJogDown.bValue = TRUE) AND (fbJogSlowToFastDlyTm.Q = TRUE) AND (bJogFast = FALSE) THEN
		tyP0935Lifter.tyMotionStd.tyBtnStop.bValue					:= FALSE;
		tyP0935Lifter.tyMotionStd.tyBtnStop.bRtLk					:= FALSE;

		fbJogSlowToFastDlyTm.IN		:= TRUE;

		diMnlLifterJogSpd	:= tyP0935Lifter.tyMotionStd.tyNumNomSpd.diValue;

		eLifterBtmAct		:= LifterActJogDown;

		IF p_eLifterBtmStat = LifterActJogDown AND p_eLifterBtmStatus = Done THEN
			eLifterBtmAct	:= LifterActIdle;
			bJogFast				:= TRUE;
		ELSIF p_eLifterBtmStatus = Error THEN
			fbJogSlowToFastDlyTm.IN	:= FALSE;
			bJogFast				:= TRUE;
		END_IF

	ELSIF (tyP0935Lifter.tyMotionStd.tyBtnJogUp.bValue = TRUE) AND (fbJogSlowToFastDlyTm.Q = FALSE) AND (bJogSlow = FALSE) THEN
		tyP0935Lifter.tyMotionStd.tyBtnStop.bValue				:= FALSE;
		tyP0935Lifter.tyMotionStd.tyBtnStop.bRtLk				:= FALSE;

		fbJogSlowToFastDlyTm.IN		:= TRUE;

		diMnlLifterJogSpd	:= tyP0935Lifter.tyMotionStd.tyNumSlwSpd.diValue;

		eLifterBtmAct		:= LifterActJogUp;

		IF p_eLifterBtmStat = LifterActJogUp AND p_eLifterBtmStatus = Done THEN
			eLifterBtmAct	:= LifterActIdle;
			bJogSlow				:= TRUE;

		ELSIF p_eLifterBtmStatus = Error THEN
			fbJogSlowToFastDlyTm.IN	:= FALSE;
			bJogSlow				:= TRUE;
		END_IF

	ELSIF (tyP0935Lifter.tyMotionStd.tyBtnJogUp.bValue = TRUE) AND (fbJogSlowToFastDlyTm.Q = TRUE) AND (bJogFast = FALSE) THEN

		tyP0935Lifter.tyMotionStd.tyBtnStop.bValue				:= FALSE;
		tyP0935Lifter.tyMotionStd.tyBtnStop.bRtLk				:= FALSE;

		fbJogSlowToFastDlyTm.IN		:= TRUE;

		diMnlLifterJogSpd	:= tyP0935Lifter.tyMotionStd.tyNumNomSpd.diValue;

		eLifterBtmAct		:= LifterActJogUp;

		IF p_eLifterBtmStat = LifterActJogUp AND p_eLifterBtmStatus = Done THEN
			eLifterBtmAct	:= LifterActIdle;
			bJogFast	:= TRUE;

		ELSIF p_eLifterBtmStatus = Error THEN
			fbJogSlowToFastDlyTm.IN	:= FALSE;
			bJogFast				:= TRUE;
		END_IF
	END_IF

	//Shutter Control
	IF tyP0935Lifter.tyInOutletShutterFB.tyBtnOpen.bRtCompl = TRUE THEN
		tyP0935Lifter.tyInOutletShutterFB.tyBtnOpen.bRtCompl	:= FALSE;

		tyP0935Lifter.tyInOutletShutterFB.tyBtnOpen.bValue	:= TRUE;
		tyP0935Lifter.tyInOutletShutterFB.tyBtnClose.bValue	:= FALSE;

	ELSIF tyP0935Lifter.tyInOutletShutterFB.tyBtnClose.bRtCompl = TRUE THEN
		tyP0935Lifter.tyInOutletShutterFB.tyBtnClose.bRtCompl	:= FALSE;

		tyP0935Lifter.tyInOutletShutterFB.tyBtnClose.bValue	:= TRUE;
		tyP0935Lifter.tyInOutletShutterFB.tyBtnOpen.bValue	:= FALSE;
	END_IF

	IF tyP0935Lifter.tyInOutletShutterFB.tyBtnOpen.bValue = TRUE THEN
		eInShutterAct	:= PneuActRet;
		eOutShutterAct	:= PneuActRet;

		IF (p_eInShutterStat = PneuActRet AND p_eInShutterStatus = Done)
			AND (p_eOutShutterStat = PneuActRet AND p_eOutShutterStatus = Done)
			THEN
			eInShutterAct	:= PneuActIdle;
			eOutShutterAct	:= PneuActIdle;
			tyP0935Lifter.tyInOutletShutterFB.tyBtnOpen.bValue	:= FALSE;
		ELSIF p_eInShutterStatus = Error OR p_eOutShutterStatus = Error THEN
			tyP0935Lifter.tyInOutletShutterFB.tyBtnOpen.bValue	:= FALSE;
		END_IF

	ELSIF tyP0935Lifter.tyInOutletShutterFB.tyBtnClose.bValue = TRUE THEN
		eInShutterAct	:= PneuActExt;
		eOutShutterAct	:= PneuActExt;
		IF (p_eInShutterStat = PneuActExt AND p_eInShutterStatus = Done)
			AND (p_eOutShutterStat = PneuActExt AND p_eOutShutterStatus = Done)
			THEN
			eInShutterAct	:= PneuActIdle;
			eOutShutterAct	:= PneuActIdle;
			tyP0935Lifter.tyInOutletShutterFB.tyBtnClose.bValue := FALSE;
		ELSIF p_eInShutterStatus = Error OR p_eOutShutterStatus = Error THEN
			tyP0935Lifter.tyInOutletShutterFB.tyBtnClose.bValue := FALSE;
		END_IF
	END_IF

END_ACTION
```

#### Act_OptP0935FBStat.st
```iecst
ACTION Act_OptP0935FBStat:

	IF p_bLifterBtmAxisErr = TRUE THEN
		tyP0935Lifter.tyMotionStd.tyStringStat.sValue	:= p_sLifterBtmAxisErrTxt;
	ELSE
		IF NOT(p_bLifterBtmJogging AND p_eLifterBtmStat = LifterActIdle) THEN
			tyP0935Lifter.tyMotionStd.tyStringStat.sValue	:= p_sLifterBtmStatTxt;
		END_IF
	END_IF

END_ACTION
```

#### Act_OptP0935Mask.st
```iecst
ACTION Act_OptP0935Mask:

	// Interlock Power
	IF p_bLifterBtmAxisErr = TRUE AND p_bLifterBtmPwrOn = FALSE THEN
		fUIInRtStatOff(ADR(tyP0935Lifter.tyMotionStd.tyBtnPwr.uiMaskRtStat));
		tyP0935Lifter.tyMotionStd.tyBtnPwr.bValue		:= FALSE;
	ELSE
		fUIInRtStatHide(ADR(tyP0935Lifter.tyMotionStd.tyBtnPwr.uiMaskRtStat));
	END_IF

	// Interlock Others Move
	IF p_bLifterBtmAxisErr = TRUE OR p_bLifterBtmPwrOn = FALSE OR
		((p_tyDI.bLifterSafetyLmtSW1 = FALSE OR p_tyDI.bLifterSafetyLmtSW2 = FALSE OR p_eDILifterSafetyStatus = Error) AND p_tyNtParamCurr.bProjLifterMagPlatform) THEN
		fUIInRtStatOff(ADR(tyP0935Lifter.tyMotionStd.tyBtnOrigin.uiMaskRtStat));
		fUIInRtStatOff(ADR(tyP0935Lifter.tyMotionStd.tyBtnMovRel.uiMaskRtStat));
		//fUIInRtStatOff(ADR(tyP0935Lifter.tyMotionStd.tyBtnJogUp.uiMaskRtStat));
		fUIInRtStatOff(ADR(tyP0935Lifter.tyMotionStd.tyBtnJogDown.uiMaskRtStat));

		IF (p_tyDI.bLifterSafetyLmtSW1 = FALSE OR p_tyDI.bLifterSafetyLmtSW2 = FALSE) AND p_tyNtParamCurr.bProjLifterMagPlatform THEN
			fUIInRtStatHide(ADR(tyP0935Lifter.tyMotionStd.tyBtnJogUp.uiMaskRtStat));
		ELSE
			fUIInRtStatOff(ADR(tyP0935Lifter.tyMotionStd.tyBtnJogUp.uiMaskRtStat));
		END_IF
	ELSE
		fUIInRtStatHide(ADR(tyP0935Lifter.tyMotionStd.tyBtnOrigin.uiMaskRtStat));
		fUIInRtStatHide(ADR(tyP0935Lifter.tyMotionStd.tyBtnMovRel.uiMaskRtStat));
		fUIInRtStatHide(ADR(tyP0935Lifter.tyMotionStd.tyBtnJogUp.uiMaskRtStat));
		fUIInRtStatHide(ADR(tyP0935Lifter.tyMotionStd.tyBtnJogDown.uiMaskRtStat));
	END_IF

	// Interlock Move Absolute
	IF p_bLifterBtmAxisErr = TRUE OR p_bLifterBtmPwrOn = FALSE OR p_bLifterBtmIsHomed = FALSE OR
		((p_tyDI.bLifterSafetyLmtSW1 = FALSE OR p_tyDI.bLifterSafetyLmtSW2 = FALSE OR p_eDILifterSafetyStatus = Error) AND p_tyNtParamCurr.bProjLifterMagPlatform) THEN

		fUIInRtStatOff(ADR(tyP0935Lifter.tyMotionStd.tyBtnMovAbs.uiMaskRtStat));

		fUIInRtStatOff(ADR(tyP0935Lifter.tyLifter.tyBtnGo.uiMaskRtStat));
		fUIInRtStatOff(ADR(tyP0935Lifter.tyLifter.tyBtnNxtSlt.uiMaskRtStat));
		fUIInRtStatOff(ADR(tyP0935Lifter.tyLifter.tyBtnPrevSlt.uiMaskRtStat));
		fUIInRtStatOff(ADR(tyP0935Lifter.tyLifter.tyBtnGoLaneA.uiMaskRtStat));
		fUIInRtStatOff(ADR(tyP0935Lifter.tyLifter.tyBtnGoLaneB.uiMaskRtStat));
		fUIInRtStatOff(ADR(tyP0935Lifter.tyLifter.tyBtnGoLaneD_G.uiMaskRtStat));
		fUIInRtStatOff(ADR(tyP0935Lifter.tyLifter.tyBtnGoLaneE_H.uiMaskRtStat));

	ELSE
		fUIInRtStatHide(ADR(tyP0935Lifter.tyMotionStd.tyBtnMovAbs.uiMaskRtStat));

		fUIInRtStatHide(ADR(tyP0935Lifter.tyLifter.tyBtnGo.uiMaskRtStat));
		fUIInRtStatHide(ADR(tyP0935Lifter.tyLifter.tyBtnNxtSlt.uiMaskRtStat));
		fUIInRtStatHide(ADR(tyP0935Lifter.tyLifter.tyBtnPrevSlt.uiMaskRtStat));
		fUIInRtStatHide(ADR(tyP0935Lifter.tyLifter.tyBtnGoLaneA.uiMaskRtStat));
		fUIInRtStatHide(ADR(tyP0935Lifter.tyLifter.tyBtnGoLaneB.uiMaskRtStat));
		fUIInRtStatHide(ADR(tyP0935Lifter.tyLifter.tyBtnGoLaneD_G.uiMaskRtStat));
		fUIInRtStatHide(ADR(tyP0935Lifter.tyLifter.tyBtnGoLaneE_H.uiMaskRtStat));

	END_IF

	//Interlock Limit Sensor
	IF tyP0935Lifter.tyMotionStd.tyBtnDownLmtSen.bValue = TRUE THEN
		fUIInRtStatOff(ADR(tyP0935Lifter.tyMotionStd.tyBtnJogDown.uiMaskRtStat));
	END_IF

	IF tyP0935Lifter.tyMotionStd.tyBtnUpLmtSen.bValue = TRUE THEN
		fUIInRtStatOff(ADR(tyP0935Lifter.tyMotionStd.tyBtnJogUp.uiMaskRtStat));
	END_IF

	// Interlock When Moving
	IF tyP0935Lifter.tyMotionStd.tyBtnOrigin.bRtCompl = TRUE THEN

		fUIInRtStatOff(ADR(tyP0935Lifter.tyMotionStd.tyBtnMovAbs.uiMaskRtStat));
		fUIInRtStatOff(ADR(tyP0935Lifter.tyMotionStd.tyBtnMovRel.uiMaskRtStat));
		fUIInRtStatOff(ADR(tyP0935Lifter.tyMotionStd.tyBtnJogUp.uiMaskRtStat));
		fUIInRtStatOff(ADR(tyP0935Lifter.tyMotionStd.tyBtnJogDown.uiMaskRtStat));

		fUIInRtStatOff(ADR(tyP0935Lifter.tyLifter.tyBtnGo.uiMaskRtStat));
		fUIInRtStatOff(ADR(tyP0935Lifter.tyLifter.tyBtnPrevSlt.uiMaskRtStat));
		fUIInRtStatOff(ADR(tyP0935Lifter.tyLifter.tyBtnNxtSlt.uiMaskRtStat));
		fUIInRtStatOff(ADR(tyP0935Lifter.tyLifter.tyBtnGoLaneA.uiMaskRtStat));
		fUIInRtStatOff(ADR(tyP0935Lifter.tyLifter.tyBtnGoLaneB.uiMaskRtStat));
		fUIInRtStatOff(ADR(tyP0935Lifter.tyLifter.tyBtnGoLaneD_G.uiMaskRtStat));
		fUIInRtStatOff(ADR(tyP0935Lifter.tyLifter.tyBtnGoLaneE_H.uiMaskRtStat));

	ELSIF tyP0935Lifter.tyMotionStd.tyBtnMovAbs.bRtCompl = TRUE THEN

		fUIInRtStatOff(ADR(tyP0935Lifter.tyMotionStd.tyBtnOrigin.uiMaskRtStat));
		fUIInRtStatOff(ADR(tyP0935Lifter.tyMotionStd.tyBtnMovRel.uiMaskRtStat));
		fUIInRtStatOff(ADR(tyP0935Lifter.tyMotionStd.tyBtnJogUp.uiMaskRtStat));
		fUIInRtStatOff(ADR(tyP0935Lifter.tyMotionStd.tyBtnJogDown.uiMaskRtStat));

		fUIInRtStatOff(ADR(tyP0935Lifter.tyLifter.tyBtnGo.uiMaskRtStat));
		fUIInRtStatOff(ADR(tyP0935Lifter.tyLifter.tyBtnPrevSlt.uiMaskRtStat));
		fUIInRtStatOff(ADR(tyP0935Lifter.tyLifter.tyBtnNxtSlt.uiMaskRtStat));
		fUIInRtStatOff(ADR(tyP0935Lifter.tyLifter.tyBtnGoLaneA.uiMaskRtStat));
		fUIInRtStatOff(ADR(tyP0935Lifter.tyLifter.tyBtnGoLaneB.uiMaskRtStat));
		fUIInRtStatOff(ADR(tyP0935Lifter.tyLifter.tyBtnGoLaneD_G.uiMaskRtStat));
		fUIInRtStatOff(ADR(tyP0935Lifter.tyLifter.tyBtnGoLaneE_H.uiMaskRtStat));

	ELSIF tyP0935Lifter.tyMotionStd.tyBtnMovRel.bRtCompl = TRUE THEN

		fUIInRtStatOff(ADR(tyP0935Lifter.tyMotionStd.tyBtnOrigin.uiMaskRtStat));
		fUIInRtStatOff(ADR(tyP0935Lifter.tyMotionStd.tyBtnMovAbs.uiMaskRtStat));
		fUIInRtStatOff(ADR(tyP0935Lifter.tyMotionStd.tyBtnJogUp.uiMaskRtStat));
		fUIInRtStatOff(ADR(tyP0935Lifter.tyMotionStd.tyBtnJogDown.uiMaskRtStat));

		fUIInRtStatOff(ADR(tyP0935Lifter.tyLifter.tyBtnGo.uiMaskRtStat));
		fUIInRtStatOff(ADR(tyP0935Lifter.tyLifter.tyBtnNxtSlt.uiMaskRtStat));
		fUIInRtStatOff(ADR(tyP0935Lifter.tyLifter.tyBtnPrevSlt.uiMaskRtStat));
		fUIInRtStatOff(ADR(tyP0935Lifter.tyLifter.tyBtnGoLaneA.uiMaskRtStat));
		fUIInRtStatOff(ADR(tyP0935Lifter.tyLifter.tyBtnGoLaneB.uiMaskRtStat));
		fUIInRtStatOff(ADR(tyP0935Lifter.tyLifter.tyBtnGoLaneD_G.uiMaskRtStat));
		fUIInRtStatOff(ADR(tyP0935Lifter.tyLifter.tyBtnGoLaneE_H.uiMaskRtStat));

	ELSIF tyP0935Lifter.tyMotionStd.tyBtnJogDown.bRtCompl = TRUE OR tyP0935Lifter.tyMotionStd.tyBtnJogDown.bValue = TRUE THEN
		fUIInRtStatOff(ADR(tyP0935Lifter.tyMotionStd.tyBtnOrigin.uiMaskRtStat));
		fUIInRtStatOff(ADR(tyP0935Lifter.tyMotionStd.tyBtnMovAbs.uiMaskRtStat));
		fUIInRtStatOff(ADR(tyP0935Lifter.tyMotionStd.tyBtnMovRel.uiMaskRtStat));
		fUIInRtStatOff(ADR(tyP0935Lifter.tyMotionStd.tyBtnJogUp.uiMaskRtStat));

		fUIInRtStatOff(ADR(tyP0935Lifter.tyLifter.tyBtnGo.uiMaskRtStat));
		fUIInRtStatOff(ADR(tyP0935Lifter.tyLifter.tyBtnNxtSlt.uiMaskRtStat));
		fUIInRtStatOff(ADR(tyP0935Lifter.tyLifter.tyBtnPrevSlt.uiMaskRtStat));
		fUIInRtStatOff(ADR(tyP0935Lifter.tyLifter.tyBtnGoLaneA.uiMaskRtStat));
		fUIInRtStatOff(ADR(tyP0935Lifter.tyLifter.tyBtnGoLaneB.uiMaskRtStat));
		fUIInRtStatOff(ADR(tyP0935Lifter.tyLifter.tyBtnGoLaneD_G.uiMaskRtStat));
		fUIInRtStatOff(ADR(tyP0935Lifter.tyLifter.tyBtnGoLaneE_H.uiMaskRtStat));

	ELSIF tyP0935Lifter.tyMotionStd.tyBtnJogUp.bRtCompl = TRUE OR tyP0935Lifter.tyMotionStd.tyBtnJogUp.bValue = TRUE THEN
		fUIInRtStatOff(ADR(tyP0935Lifter.tyMotionStd.tyBtnOrigin.uiMaskRtStat));
		fUIInRtStatOff(ADR(tyP0935Lifter.tyMotionStd.tyBtnMovAbs.uiMaskRtStat));
		fUIInRtStatOff(ADR(tyP0935Lifter.tyMotionStd.tyBtnMovRel.uiMaskRtStat));
		fUIInRtStatOff(ADR(tyP0935Lifter.tyMotionStd.tyBtnJogDown.uiMaskRtStat));

		fUIInRtStatOff(ADR(tyP0935Lifter.tyLifter.tyBtnGo.uiMaskRtStat));
		fUIInRtStatOff(ADR(tyP0935Lifter.tyLifter.tyBtnNxtSlt.uiMaskRtStat));
		fUIInRtStatOff(ADR(tyP0935Lifter.tyLifter.tyBtnPrevSlt.uiMaskRtStat));
		fUIInRtStatOff(ADR(tyP0935Lifter.tyLifter.tyBtnGoLaneA.uiMaskRtStat));
		fUIInRtStatOff(ADR(tyP0935Lifter.tyLifter.tyBtnGoLaneB.uiMaskRtStat));
		fUIInRtStatOff(ADR(tyP0935Lifter.tyLifter.tyBtnGoLaneD_G.uiMaskRtStat));
		fUIInRtStatOff(ADR(tyP0935Lifter.tyLifter.tyBtnGoLaneE_H.uiMaskRtStat));

	ELSIF tyP0935Lifter.tyLifter.tyBtnGo.bRtCompl = TRUE THEN
		fUIInRtStatOff(ADR(tyP0935Lifter.tyMotionStd.tyBtnOrigin.uiMaskRtStat));
		fUIInRtStatOff(ADR(tyP0935Lifter.tyMotionStd.tyBtnMovAbs.uiMaskRtStat));
		fUIInRtStatOff(ADR(tyP0935Lifter.tyMotionStd.tyBtnMovRel.uiMaskRtStat));
		fUIInRtStatOff(ADR(tyP0935Lifter.tyMotionStd.tyBtnJogUp.uiMaskRtStat));
		fUIInRtStatOff(ADR(tyP0935Lifter.tyMotionStd.tyBtnJogDown.uiMaskRtStat));

		fUIInRtStatOff(ADR(tyP0935Lifter.tyLifter.tyBtnNxtSlt.uiMaskRtStat));
		fUIInRtStatOff(ADR(tyP0935Lifter.tyLifter.tyBtnPrevSlt.uiMaskRtStat));
		fUIInRtStatOff(ADR(tyP0935Lifter.tyLifter.tyBtnGoLaneA.uiMaskRtStat));
		fUIInRtStatOff(ADR(tyP0935Lifter.tyLifter.tyBtnGoLaneB.uiMaskRtStat));
		fUIInRtStatOff(ADR(tyP0935Lifter.tyLifter.tyBtnGoLaneD_G.uiMaskRtStat));
		fUIInRtStatOff(ADR(tyP0935Lifter.tyLifter.tyBtnGoLaneE_H.uiMaskRtStat));

	ELSIF tyP0935Lifter.tyLifter.tyBtnNxtSlt.bRtCompl = TRUE THEN
		fUIInRtStatOff(ADR(tyP0935Lifter.tyMotionStd.tyBtnOrigin.uiMaskRtStat));
		fUIInRtStatOff(ADR(tyP0935Lifter.tyMotionStd.tyBtnMovAbs.uiMaskRtStat));
		fUIInRtStatOff(ADR(tyP0935Lifter.tyMotionStd.tyBtnMovRel.uiMaskRtStat));
		fUIInRtStatOff(ADR(tyP0935Lifter.tyMotionStd.tyBtnJogUp.uiMaskRtStat));
		fUIInRtStatOff(ADR(tyP0935Lifter.tyMotionStd.tyBtnJogDown.uiMaskRtStat));

		fUIInRtStatOff(ADR(tyP0935Lifter.tyLifter.tyBtnGo.uiMaskRtStat));
		fUIInRtStatOff(ADR(tyP0935Lifter.tyLifter.tyBtnPrevSlt.uiMaskRtStat));
		fUIInRtStatOff(ADR(tyP0935Lifter.tyLifter.tyBtnGoLaneA.uiMaskRtStat));
		fUIInRtStatOff(ADR(tyP0935Lifter.tyLifter.tyBtnGoLaneB.uiMaskRtStat));
		fUIInRtStatOff(ADR(tyP0935Lifter.tyLifter.tyBtnGoLaneD_G.uiMaskRtStat));
		fUIInRtStatOff(ADR(tyP0935Lifter.tyLifter.tyBtnGoLaneE_H.uiMaskRtStat));

	ELSIF tyP0935Lifter.tyLifter.tyBtnPrevSlt.bRtCompl = TRUE THEN
		fUIInRtStatOff(ADR(tyP0935Lifter.tyMotionStd.tyBtnOrigin.uiMaskRtStat));
		fUIInRtStatOff(ADR(tyP0935Lifter.tyMotionStd.tyBtnMovAbs.uiMaskRtStat));
		fUIInRtStatOff(ADR(tyP0935Lifter.tyMotionStd.tyBtnMovRel.uiMaskRtStat));
		fUIInRtStatOff(ADR(tyP0935Lifter.tyMotionStd.tyBtnJogUp.uiMaskRtStat));
		fUIInRtStatOff(ADR(tyP0935Lifter.tyMotionStd.tyBtnJogDown.uiMaskRtStat));

		fUIInRtStatOff(ADR(tyP0935Lifter.tyLifter.tyBtnGo.uiMaskRtStat));
		fUIInRtStatOff(ADR(tyP0935Lifter.tyLifter.tyBtnNxtSlt.uiMaskRtStat));
		fUIInRtStatOff(ADR(tyP0935Lifter.tyLifter.tyBtnGoLaneA.uiMaskRtStat));
		fUIInRtStatOff(ADR(tyP0935Lifter.tyLifter.tyBtnGoLaneB.uiMaskRtStat));
		fUIInRtStatOff(ADR(tyP0935Lifter.tyLifter.tyBtnGoLaneD_G.uiMaskRtStat));
		fUIInRtStatOff(ADR(tyP0935Lifter.tyLifter.tyBtnGoLaneE_H.uiMaskRtStat));

	ELSIF tyP0935Lifter.tyLifter.tyBtnGoLaneA.bRtCompl = TRUE THEN
		fUIInRtStatOff(ADR(tyP0935Lifter.tyMotionStd.tyBtnOrigin.uiMaskRtStat));
		fUIInRtStatOff(ADR(tyP0935Lifter.tyMotionStd.tyBtnMovAbs.uiMaskRtStat));
		fUIInRtStatOff(ADR(tyP0935Lifter.tyMotionStd.tyBtnMovRel.uiMaskRtStat));
		fUIInRtStatOff(ADR(tyP0935Lifter.tyMotionStd.tyBtnJogUp.uiMaskRtStat));
		fUIInRtStatOff(ADR(tyP0935Lifter.tyMotionStd.tyBtnJogDown.uiMaskRtStat));

		fUIInRtStatOff(ADR(tyP0935Lifter.tyLifter.tyBtnGo.uiMaskRtStat));
		fUIInRtStatOff(ADR(tyP0935Lifter.tyLifter.tyBtnNxtSlt.uiMaskRtStat));
		fUIInRtStatOff(ADR(tyP0935Lifter.tyLifter.tyBtnPrevSlt.uiMaskRtStat));
		fUIInRtStatOff(ADR(tyP0935Lifter.tyLifter.tyBtnGoLaneB.uiMaskRtStat));
		fUIInRtStatOff(ADR(tyP0935Lifter.tyLifter.tyBtnGoLaneE_H.uiMaskRtStat));

	ELSIF tyP0935Lifter.tyLifter.tyBtnGoLaneB.bRtCompl = TRUE THEN
		fUIInRtStatOff(ADR(tyP0935Lifter.tyMotionStd.tyBtnOrigin.uiMaskRtStat));
		fUIInRtStatOff(ADR(tyP0935Lifter.tyMotionStd.tyBtnMovAbs.uiMaskRtStat));
		fUIInRtStatOff(ADR(tyP0935Lifter.tyMotionStd.tyBtnMovRel.uiMaskRtStat));
		fUIInRtStatOff(ADR(tyP0935Lifter.tyMotionStd.tyBtnJogUp.uiMaskRtStat));
		fUIInRtStatOff(ADR(tyP0935Lifter.tyMotionStd.tyBtnJogDown.uiMaskRtStat));

		fUIInRtStatOff(ADR(tyP0935Lifter.tyLifter.tyBtnGo.uiMaskRtStat));
		fUIInRtStatOff(ADR(tyP0935Lifter.tyLifter.tyBtnNxtSlt.uiMaskRtStat));
		fUIInRtStatOff(ADR(tyP0935Lifter.tyLifter.tyBtnPrevSlt.uiMaskRtStat));
		fUIInRtStatOff(ADR(tyP0935Lifter.tyLifter.tyBtnGoLaneA.uiMaskRtStat));
		fUIInRtStatOff(ADR(tyP0935Lifter.tyLifter.tyBtnGoLaneD_G.uiMaskRtStat));

	END_IF

	//Axis Error
	IF tyP0935Lifter.tyMotionStd.tyBtnPwr.bRtCompl = TRUE THEN
		fUIInRtStatOff(ADR(tyP0935Lifter.tyMotionStd.tyBtnRst.uiMaskRtStat));
	ELSE
		fUIInRtStatHide(ADR(tyP0935Lifter.tyMotionStd.tyBtnRst.uiMaskRtStat));
	END_IF

	//Next Slot
	IF p_diLifterBtmCurrSltA >= p_tyProdRcpCurrRcp0.diMaxSltValue THEN
		fUIInRtStatOff(ADR(tyP0935Lifter.tyLifter.tyBtnNxtSlt.uiMaskRtStat));
	END_IF

	//Previous Slot
	IF p_diLifterBtmCurrSltA <= p_tyProdRcpCurrRcp0.diMinSltValue THEN
		fUIInRtStatOff(ADR(tyP0935Lifter.tyLifter.tyBtnPrevSlt.uiMaskRtStat));
	END_IF

END_ACTION
```
